LIN {X 0,Y 336.735,Z 952.723,A -85,B 0,C 180,E1 12207.175,E2 12207.175} C_VEL
LIN {X 0,Y 325.926,Z 967.689,A -85,B 0,C 180,E1 12204.691,E2 12204.691} C_VEL
LIN {X 0,Y 313.476,Z 984.143,A -85,B 0,C 180,E1 12201.395,E2 12201.395} C_VEL
LIN {X 0,Y 302.068,Z 998.366,A -85,B 0,C 180,E1 12197.857,E2 12197.857} C_VEL
LIN {X 0,Y 292.752,Z 1009.779,A -85,B 0,C 180,E1 12194.441,E2 12194.441} C_VEL
LIN {X 0,Y 282.433,Z 1022.378,A -85,B 0,C 180,E1 12189.85,E2 12189.85} C_VEL
LIN {X 0,Y 274.164,Z 1032.514,A -85,B 0,C 180,E1 12185.186,E2 12185.186} C_VEL
LIN {X 0,Y 268.041,Z 1040.43,A -85,B 0,C 180,E1 12180.734,E2 12180.734} C_VEL
LIN {X 0,Y 262.356,Z 1048.512,A -85,B 0,C 180,E1 12175.027,E2 12175.027} C_VEL
LIN {X 0,Y 258.976,Z 1054.032,A -85,B 0,C 180,E1 12169.862,E2 12169.862} C_VEL
LIN {X 0,Y 257.187,Z 1057.754,A -85,B 0,C 180,E1 12165.33,E2 12165.33} C_VEL
LIN {X 0,Y 256.255,Z 1060.464,A -85,B 0,C 180,E1 12160.795,E2 12160.795} C_VEL
LIN {X 0,Y 255.945,Z 1062.179,A -85,B 0,C 180,E1 12156.28,E2 12156.28} C_VEL
LIN {X 0,Y 255.908,Z 1062.926,A -85,B 0,C 180,E1 12151.567,E2 12151.567} C_VEL
LIN {X 0,Y 255.912,Z 1062.587,A -85,B 0,C 180,E1 12146.864,E2 12146.864} C_VEL
LIN {X 0,Y 256.04,Z 1060.822,A -85,B 0,C 180,E1 12141.692,E2 12141.692} C_VEL
LIN {X 0,Y 256.6,Z 1058.068,A -85,B 0,C 180,E1 12136.938,E2 12136.938} C_VEL
LIN {X 0,Y 257.893,Z 1054.397,A -85,B 0,C 180,E1 12132.397,E2 12132.397} C_VEL
LIN {X 0,Y 260.268,Z 1049.406,A -85,B 0,C 180,E1 12127.646,E2 12127.646} C_VEL
LIN {X 0,Y 264.917,Z 1041.534,A -85,B 0,C 180,E1 12121.85,E2 12121.85} C_VEL
LIN {X 0,Y 270.469,Z 1033.203,A -85,B 0,C 180,E1 12117.055,E2 12117.055} C_VEL
LIN {X 0,Y 277.094,Z 1023.98,A -85,B 0,C 180,E1 12112.683,E2 12112.683} C_VEL
LIN {X 0,Y 286.962,Z 1010.708,A -85,B 0,C 180,E1 12107.621,E2 12107.621} C_VEL
LIN {X 0,Y 295.813,Z 998.833,A -85,B 0,C 180,E1 12103.949,E2 12103.949} C_VEL
LIN {X 0,Y 306.537,Z 984.365,A -85,B 0,C 180,E1 12100.23,E2 12100.23} C_VEL
LIN {X 0,Y 317.721,Z 968.541,A -85,B 0,C 180,E1 12096.932,E2 12096.932} C_VEL
LIN {X 0,Y 327.989,Z 953.379,A -85,B 0,C 180,E1 12094.295,E2 12094.295} C_VEL
LIN {X 0,Y 339.558,Z 935.432,A -85,B 0,C 180,E1 12091.679,E2 12091.679} C_VEL
LIN {X 0,Y 351.058,Z 915.947,A -85,B 0,C 180,E1 12089.361,E2 12089.361} C_VEL
LIN {X 0,Y 360.57,Z 898.596,A -85,B 0,C 180,E1 12087.626,E2 12087.626} C_VEL
LIN {X 0,Y 371.142,Z 877.701,A -85,B 0,C 180,E1 12085.866,E2 12085.866} C_VEL
LIN {X 0,Y 381.228,Z 855.132,A -85,B 0,C 180,E1 12084.317,E2 12084.317} C_VEL
LIN {X 0,Y 388.946,Z 835.881,A -85,B 0,C 180,E1 12083.213,E2 12083.213} C_VEL
LIN {X 0,Y 397.181,Z 812.804,A -85,B 0,C 180,E1 12082.116,E2 12082.116} C_VEL
LIN {X 0,Y 404.562,Z 787.996,A -85,B 0,C 180,E1 12081.181,E2 12081.181} C_VEL
LIN {X 0,Y 409.672,Z 767.607,A -85,B 0,C 180,E1 12080.56,E2 12080.56} C_VEL
LIN {X 0,Y 414.754,Z 742.941,A -85,B 0,C 180,E1 12079.967,E2 12079.967} C_VEL
LIN {X 0,Y 418.524,Z 716.56,A -85,B 0,C 180,E1 12079.475,E2 12079.475} C_VEL
LIN {X 0,Y 437.682,Z 506.178,A -85,B 0,C 180,E1 12076.237,E2 12076.237} C_VEL
LIN {X 0,Y 432.715,Z 497.153,A -85,B 0,C 180,E1 12073.496,E2 12073.496} C_VEL
LIN {X 0,Y 428.974,Z 490.578,A -85,B 0,C 180,E1 12071.019,E2 12071.019} C_VEL
LIN {X 0,Y 426.712,Z 486.682,A -85,B 0,C 180,E1 12069.237,E2 12069.237} C_VEL
LIN {X 0,Y 424.543,Z 482.925,A -85,B 0,C 180,E1 12067.171,E2 12067.171} C_VEL
LIN {X 0,Y 422.269,Z 478.811,A -85,B 0,C 180,E1 12064.21,E2 12064.21} C_VEL
LIN {X 0,Y 420.494,Z 475.74,A -85,B 0,C 180,E1 12058.501,E2 12058.501} C_VEL
LIN {X 0,Y 420.904,Z 477.2,A -85,B 0,C 180,E1 12055.367,E2 12055.367} C_VEL
LIN {X 0,Y 422.548,Z 479.254,A -85,B 0,C 180,E1 12052.18,E2 12052.18} C_VEL
LIN {X 0,Y 425.298,Z 484.171,A -85,B 0,C 180,E1 12048.885,E2 12048.885} C_VEL
LIN {X 0,Y 428.058,Z 488.972,A -85,B 0,C 180,E1 12046.492,E2 12046.492} C_VEL
LIN {X 0,Y 432.057,Z 495.823,A -85,B 0,C 180,E1 12043.738,E2 12043.738} C_VEL
LIN {X 0,Y 436.565,Z 504.122,A -85,B 0,C 180,E1 12041.159,E2 12041.159} C_VEL
LIN {X 0,Y 437.639,Z 506.238,A -85,B 0,C 180,E1 12040.598,E2 12040.598} C_VEL
LIN {X 0,Y 418.656,Z 714.21,A -85,B 0,C 180,E1 12037.403,E2 12037.403} C_VEL
LIN {X 0,Y 414.746,Z 741.081,A -85,B 0,C 180,E1 12036.896,E2 12036.896} C_VEL
LIN {X 0,Y 409.832,Z 764.962,A -85,B 0,C 180,E1 12036.307,E2 12036.307} C_VEL
LIN {X 0,Y 404.496,Z 786.334,A -85,B 0,C 180,E1 12035.63,E2 12035.63} C_VEL
LIN {X 0,Y 396.755,Z 812.006,A -85,B 0,C 180,E1 12034.619,E2 12034.619} C_VEL
LIN {X 0,Y 389.497,Z 832.399,A -85,B 0,C 180,E1 12033.627,E2 12033.627} C_VEL
LIN {X 0,Y 381.614,Z 852.091,A -85,B 0,C 180,E1 12032.489,E2 12032.489} C_VEL
LIN {X 0,Y 371.507,Z 874.688,A -85,B 0,C 180,E1 12030.918,E2 12030.918} C_VEL
LIN {X 0,Y 361.031,Z 895.39,A -85,B 0,C 180,E1 12029.154,E2 12029.154} C_VEL
LIN {X 0,Y 351.198,Z 913.285,A -85,B 0,C 180,E1 12027.343,E2 12027.343} C_VEL
LIN {X 0,Y 338.52,Z 934.435,A -85,B 0,C 180,E1 12024.755,E2 12024.755} C_VEL
LIN {X 0,Y 328.196,Z 950.374,A -85,B 0,C 180,E1 12022.384,E2 12022.384} C_VEL
LIN {X 0,Y 318.152,Z 965.114,A -85,B 0,C 180,E1 12019.791,E2 12019.791} C_VEL
LIN {X 0,Y 305.579,Z 982.616,A -85,B 0,C 180,E1 12016.043,E2 12016.043} C_VEL
LIN {X 0,Y 296.17,Z 995.232,A -85,B 0,C 180,E1 12012.733,E2 12012.733} C_VEL
LIN {X 0,Y 286.879,Z 1007.573,A -85,B 0,C 180,E1 12008.856,E2 12008.856} C_VEL
LIN {X 0,Y 277.456,Z 1019.987,A -85,B 0,C 180,E1 12004.017,E2 12004.017} C_VEL
LIN {X 0,Y 271.095,Z 1028.659,A -85,B 0,C 180,E1 11999.863,E2 11999.863} C_VEL
LIN {X 0,Y 265.325,Z 1037.081,A -85,B 0,C 180,E1 11994.966,E2 11994.966} C_VEL
LIN {X 0,Y 260.629,Z 1044.701,A -85,B 0,C 180,E1 11989.265,E2 11989.265} C_VEL
LIN {X 0,Y 258.12,Z 1049.684,A -85,B 0,C 180,E1 11984.432,E2 11984.432} C_VEL
LIN {X 0,Y 256.696,Z 1053.442,A -85,B 0,C 180,E1 11979.642,E2 11979.642} C_VEL
LIN {X 0,Y 256.042,Z 1056.374,A -85,B 0,C 180,E1 11974.255,E2 11974.255} C_VEL
LIN {X 0,Y 255.923,Z 1057.688,A -85,B 0,C 180,E1 11969.328,E2 11969.328} C_VEL
LIN {X 0,Y 255.916,Z 1057.898,A -85,B 0,C 180,E1 11964.844,E2 11964.844} C_VEL
LIN {X 0,Y 256.005,Z 1057.204,A -85,B 0,C 180,E1 11960.558,E2 11960.558} C_VEL
LIN {X 0,Y 256.395,Z 1055.589,A -85,B 0,C 180,E1 11956.181,E2 11956.181} C_VEL
LIN {X 0,Y 257.427,Z 1052.964,A -85,B 0,C 180,E1 11951.662,E2 11951.662} C_VEL
LIN {X 0,Y 259.468,Z 1049.079,A -85,B 0,C 180,E1 11946.855,E2 11946.855} C_VEL
LIN {X 0,Y 263.498,Z 1042.971,A -85,B 0,C 180,E1 11941.189,E2 11941.189} C_VEL
LIN {X 0,Y 269.013,Z 1035.478,A -85,B 0,C 180,E1 11935.983,E2 11935.983} C_VEL
LIN {X 0,Y 275.246,Z 1027.677,A -85,B 0,C 180,E1 11931.597,E2 11931.597} C_VEL
LIN {X 0,Y 284.248,Z 1016.9,A -85,B 0,C 180,E1 11926.69,E2 11926.69} C_VEL
LIN {X 0,Y 294.039,Z 1005.111,A -85,B 0,C 180,E1 11922.446,E2 11922.446} C_VEL
LIN {X 0,Y 303.724,Z 993.402,A -85,B 0,C 180,E1 11918.961,E2 11918.961} C_VEL
LIN {X 0,Y 316.508,Z 977.44,A -85,B 0,C 180,E1 11915.094,E2 11915.094} C_VEL
LIN {X 0,Y 327.49,Z 962.979,A -85,B 0,C 180,E1 11912.25,E2 11912.25} C_VEL
LIN {X 0,Y 338.542,Z 947.715,A -85,B 0,C 180,E1 11909.735,E2 11909.735} C_VEL
LIN {X 0,Y 352.289,Z 927.25,A -85,B 0,C 180,E1 11906.974,E2 11906.974} C_VEL
LIN {X 0,Y 362.606,Z 910.598,A -85,B 0,C 180,E1 11905.129,E2 11905.129} C_VEL
LIN {X 0,Y 372.78,Z 892.869,A -85,B 0,C 180,E1 11903.462,E2 11903.462} C_VEL
LIN {X 0,Y 384.665,Z 869.928,A -85,B 0,C 180,E1 11901.678,E2 11901.678} C_VEL
LIN {X 0,Y 393.697,Z 850.323,A -85,B 0,C 180,E1 11900.42,E2 11900.42} C_VEL
LIN {X 0,Y 402.231,Z 829.664,A -85,B 0,C 180,E1 11899.306,E2 11899.306} C_VEL
LIN {X 0,Y 411.481,Z 803.641,A -85,B 0,C 180,E1 11898.174,E2 11898.174} C_VEL
LIN {X 0,Y 417.687,Z 783.031,A -85,B 0,C 180,E1 11897.455,E2 11897.455} C_VEL
LIN {X 0,Y 423.053,Z 761.928,A -85,B 0,C 180,E1 11896.847,E2 11896.847} C_VEL
LIN {X 0,Y 428.658,Z 733.815,A -85,B 0,C 180,E1 11896.229,E2 11896.229} C_VEL
LIN {X 0,Y 431.2,Z 716.612,A -85,B 0,C 180,E1 11895.925,E2 11895.925} C_VEL
LIN {X 0,Y 431.767,Z 709.092,A -85,B 0,C 180,E1 11895.676,E2 11895.676} C_VEL
LIN {X 0,Y 431.958,Z 689.518,A -85,B 0,C 180,E1 11894.578,E2 11894.578} C_VEL
LIN {X 0,Y 432.363,Z 683.031,A -85,B 0,C 180,E1 11894.388,E2 11894.388} C_VEL
LIN {X 0,Y 448.077,Z 521.035,A -85,B 0,C 180,E1 11891.978,E2 11891.978} C_VEL
LIN {X 0,Y 444.633,Z 514.491,A -85,B 0,C 180,E1 11889.449,E2 11889.449} C_VEL
LIN {X 0,Y 442.12,Z 509.966,A -85,B 0,C 180,E1 11887.145,E2 11887.145} C_VEL
LIN {X 0,Y 440.219,Z 506.351,A -85,B 0,C 180,E1 11884.821,E2 11884.821} C_VEL
LIN {X 0,Y 438.336,Z 501.994,A -85,B 0,C 180,E1 11880.392,E2 11880.392} C_VEL
LIN {X 0,Y 438.418,Z 502.124,A -85,B 0,C 180,E1 11876.339,E2 11876.339} C_VEL
LIN {X 0,Y 440.195,Z 506.386,A -85,B 0,C 180,E1 11872.298,E2 11872.298} C_VEL
LIN {X 0,Y 441.119,Z 508.161,A -85,B 0,C 180,E1 11871.068,E2 11871.068} C_VEL
LIN {X 0,Y 443.036,Z 511.664,A -85,B 0,C 180,E1 11869.037,E2 11869.037} C_VEL
LIN {X 0,Y 445.731,Z 516.615,A -85,B 0,C 180,E1 11866.773,E2 11866.773} C_VEL
LIN {X 0,Y 448.131,Z 521.442,A -85,B 0,C 180,E1 11865.061,E2 11865.061} C_VEL
LIN {X 0,Y 428.944,Z 716.865,A -85,B 0,C 180,E1 11862.164,E2 11862.164} C_VEL
LIN {X 0,Y 424.778,Z 743.872,A -85,B 0,C 180,E1 11861.688,E2 11861.688} C_VEL
LIN {X 0,Y 419.625,Z 767.55,A -85,B 0,C 180,E1 11861.159,E2 11861.159} C_VEL
LIN {X 0,Y 414.229,Z 787.872,A -85,B 0,C 180,E1 11860.595,E2 11860.595} C_VEL
LIN {X 0,Y 406.633,Z 812.077,A -85,B 0,C 180,E1 11859.757,E2 11859.757} C_VEL
LIN {X 0,Y 398.007,Z 834.964,A -85,B 0,C 180,E1 11858.755,E2 11858.755} C_VEL
LIN {X 0,Y 389.986,Z 853.879,A -85,B 0,C 180,E1 11857.754,E2 11857.754} C_VEL
LIN {X 0,Y 380.517,Z 873.928,A -85,B 0,C 180,E1 11856.501,E2 11856.501} C_VEL
LIN {X 0,Y 368.599,Z 896.322,A -85,B 0,C 180,E1 11854.793,E2 11854.793} C_VEL
LIN {X 0,Y 358.091,Z 914.215,A -85,B 0,C 180,E1 11853.142,E2 11853.142} C_VEL
LIN {X 0,Y 346.16,Z 933.011,A -85,B 0,C 180,E1 11851.071,E2 11851.071} C_VEL
LIN {X 0,Y 332.963,Z 951.98,A -85,B 0,C 180,E1 11848.498,E2 11848.498} C_VEL
LIN {X 0,Y 321.859,Z 966.938,A -85,B 0,C 180,E1 11846.043,E2 11846.043} C_VEL
LIN {X 0,Y 309.548,Z 982.746,A -85,B 0,C 180,E1 11842.925,E2 11842.925} C_VEL
LIN {X 0,Y 297.095,Z 997.78,A -85,B 0,C 180,E1 11839.222,E2 11839.222} C_VEL
LIN {X 0,Y 287.355,Z 1009.241,A -85,B 0,C 180,E1 11835.791,E2 11835.791} C_VEL
LIN {X 0,Y 276.791,Z 1021.62,A -85,B 0,C 180,E1 11831.289,E2 11831.289} C_VEL
LIN {X 0,Y 267.758,Z 1032.109,A -85,B 0,C 180,E1 11826.424,E2 11826.424} C_VEL
LIN {X 0,Y 261.207,Z 1040.066,A -85,B 0,C 180,E1 11821.888,E2 11821.888} C_VEL
LIN {X 0,Y 255.228,Z 1048.032,A -85,B 0,C 180,E1 11816.215,E2 11816.215} C_VEL
LIN {X 0,Y 251.264,Z 1053.993,A -85,B 0,C 180,E1 11810.499,E2 11810.499} C_VEL
LIN {X 0,Y 249.25,Z 1057.866,A -85,B 0,C 180,E1 11805.591,E2 11805.591} C_VEL
LIN {X 0,Y 248.234,Z 1060.661,A -85,B 0,C 180,E1 11800.629,E2 11800.629} C_VEL
LIN {X 0,Y 247.917,Z 1062.458,A -85,B 0,C 180,E1 11795.323,E2 11795.323} C_VEL
LIN {X 0,Y 247.927,Z 1062.847,A -85,B 0,C 180,E1 11790.231,E2 11790.231} C_VEL
LIN {X 0,Y 247.909,Z 1062.171,A -85,B 0,C 180,E1 11785.605,E2 11785.605} C_VEL
LIN {X 0,Y 248.062,Z 1060.606,A -85,B 0,C 180,E1 11781.189,E2 11781.189} C_VEL
LIN {X 0,Y 248.68,Z 1057.958,A -85,B 0,C 180,E1 11776.514,E2 11776.514} C_VEL
LIN {X 0,Y 250.09,Z 1054.277,A -85,B 0,C 180,E1 11771.829,E2 11771.829} C_VEL
LIN {X 0,Y 252.654,Z 1049.276,A -85,B 0,C 180,E1 11766.934,E2 11766.934} C_VEL
LIN {X 0,Y 257.86,Z 1041.018,A -85,B 0,C 180,E1 11760.748,E2 11760.748} C_VEL
LIN {X 0,Y 263.472,Z 1033.085,A -85,B 0,C 180,E1 11756.092,E2 11756.092} C_VEL
LIN {X 0,Y 270.136,Z 1024.272,A -85,B 0,C 180,E1 11751.82,E2 11751.82} C_VEL
LIN {X 0,Y 279.766,Z 1011.932,A -85,B 0,C 180,E1 11746.95,E2 11746.95} C_VEL
LIN {X 0,Y 289.577,Z 999.267,A -85,B 0,C 180,E1 11742.944,E2 11742.944} C_VEL
LIN {X 0,Y 299.517,Z 986.31,A -85,B 0,C 180,E1 11739.543,E2 11739.543} C_VEL
LIN {X 0,Y 312.183,Z 969.143,A -85,B 0,C 180,E1 11735.872,E2 11735.872} C_VEL
LIN {X 0,Y 322.736,Z 954.047,A -85,B 0,C 180,E1 11733.228,E2 11733.228} C_VEL
LIN {X 0,Y 333.46,Z 937.893,A -85,B 0,C 180,E1 11730.847,E2 11730.847} C_VEL
LIN {X 0,Y 346.371,Z 916.849,A -85,B 0,C 180,E1 11728.303,E2 11728.303} C_VEL
LIN {X 0,Y 356.09,Z 899.594,A -85,B 0,C 180,E1 11726.577,E2 11726.577} C_VEL
LIN {X 0,Y 365.881,Z 880.749,A -85,B 0,C 180,E1 11724.98,E2 11724.98} C_VEL
LIN {X 0,Y 377.235,Z 856.32,A -85,B 0,C 180,E1 11723.285,E2 11723.285} C_VEL
LIN {X 0,Y 385.404,Z 836.41,A -85,B 0,C 180,E1 11722.151,E2 11722.151} C_VEL
LIN {X 0,Y 393.112,Z 815.314,A -85,B 0,C 180,E1 11721.154,E2 11721.154} C_VEL
LIN {X 0,Y 401.068,Z 789.631,A -85,B 0,C 180,E1 11720.177,E2 11720.177} C_VEL
LIN {X 0,Y 406.458,Z 768.682,A -85,B 0,C 180,E1 11719.54,E2 11719.54} C_VEL
LIN {X 0,Y 411.248,Z 746.109,A -85,B 0,C 180,E1 11718.997,E2 11718.997} C_VEL
LIN {X 0,Y 415.567,Z 717.905,A -85,B 0,C 180,E1 11718.465,E2 11718.465} C_VEL
LIN {X 0,Y 425.663,Z 609.9,A -85,B 0,C 180,E1 11716.798,E2 11716.798} C_VEL
LIN {X 0,Y 434.788,Z 511.445,A -85,B 0,C 180,E1 11715.301,E2 11715.301} C_VEL
LIN {X 0,Y 430.262,Z 502.918,A -85,B 0,C 180,E1 11712.618,E2 11712.618} C_VEL
LIN {X 0,Y 426.048,Z 495.294,A -85,B 0,C 180,E1 11709.524,E2 11709.524} C_VEL
LIN {X 0,Y 423.304,Z 490.638,A -85,B 0,C 180,E1 11706.919,E2 11706.919} C_VEL
LIN {X 0,Y 421.203,Z 486.697,A -85,B 0,C 180,E1 11704.084,E2 11704.084} C_VEL
LIN {X 0,Y 419.519,Z 483.683,A -85,B 0,C 180,E1 11698.498,E2 11698.498} C_VEL
LIN {X 0,Y 420.018,Z 485.34,A -85,B 0,C 180,E1 11695.084,E2 11695.084} C_VEL
LIN {X 0,Y 421.476,Z 487.179,A -85,B 0,C 180,E1 11692.297,E2 11692.297} C_VEL
LIN {X 0,Y 424.108,Z 492.007,A -85,B 0,C 180,E1 11689.059,E2 11689.059} C_VEL
LIN {X 0,Y 426.729,Z 496.681,A -85,B 0,C 180,E1 11686.725,E2 11686.725} C_VEL
LIN {X 0,Y 430.589,Z 503.495,A -85,B 0,C 180,E1 11683.993,E2 11683.993} C_VEL
LIN {X 0,Y 434.769,Z 511.39,A -85,B 0,C 180,E1 11681.53,E2 11681.53} C_VEL
LIN {X 0,Y 415.857,Z 714.241,A -85,B 0,C 180,E1 11678.435,E2 11678.435} C_VEL
LIN {X 0,Y 411.897,Z 741.045,A -85,B 0,C 180,E1 11677.936,E2 11677.936} C_VEL
LIN {X 0,Y 406.891,Z 765,A -85,B 0,C 180,E1 11677.356,E2 11677.356} C_VEL
LIN {X 0,Y 401.415,Z 786.552,A -85,B 0,C 180,E1 11676.684,E2 11676.684} C_VEL
LIN {X 0,Y 393.637,Z 811.908,A -85,B 0,C 180,E1 11675.701,E2 11675.701} C_VEL
LIN {X 0,Y 386.006,Z 832.931,A -85,B 0,C 180,E1 11674.692,E2 11674.692} C_VEL
LIN {X 0,Y 377.974,Z 852.577,A -85,B 0,C 180,E1 11673.567,E2 11673.567} C_VEL
LIN {X 0,Y 367.135,Z 876.128,A -85,B 0,C 180,E1 11671.934,E2 11671.934} C_VEL
LIN {X 0,Y 356.959,Z 895.772,A -85,B 0,C 180,E1 11670.267,E2 11670.267} C_VEL
LIN {X 0,Y 347.096,Z 913.3,A -85,B 0,C 180,E1 11668.505,E2 11668.505} C_VEL
LIN {X 0,Y 334.232,Z 934.247,A -85,B 0,C 180,E1 11665.962,E2 11665.962} C_VEL
LIN {X 0,Y 323.726,Z 950.04,A -85,B 0,C 180,E1 11663.627,E2 11663.627} C_VEL
LIN {X 0,Y 313.458,Z 964.67,A -85,B 0,C 180,E1 11661.067,E2 11661.067} C_VEL
LIN {X 0,Y 301.039,Z 981.477,A -85,B 0,C 180,E1 11657.507,E2 11657.507} C_VEL
LIN {X 0,Y 290.692,Z 994.835,A -85,B 0,C 180,E1 11654.012,E2 11654.012} C_VEL
LIN {X 0,Y 281.403,Z 1006.657,A -85,B 0,C 180,E1 11650.292,E2 11650.292} C_VEL
LIN {X 0,Y 270.976,Z 1019.83,A -85,B 0,C 180,E1 11645.144,E2 11645.144} C_VEL
LIN {X 0,Y 263.942,Z 1028.944,A -85,B 0,C 180,E1 11640.689,E2 11640.689} C_VEL
LIN {X 0,Y 257.713,Z 1037.593,A -85,B 0,C 180,E1 11635.509,E2 11635.509} C_VEL
LIN {X 0,Y 252.903,Z 1044.938,A -85,B 0,C 180,E1 11629.784,E2 11629.784} C_VEL
LIN {X 0,Y 250.347,Z 1049.677,A -85,B 0,C 180,E1 11625.047,E2 11625.047} C_VEL
LIN {X 0,Y 248.806,Z 1053.4,A -85,B 0,C 180,E1 11620.185,E2 11620.185} C_VEL
LIN {X 0,Y 248.065,Z 1056.377,A -85,B 0,C 180,E1 11614.624,E2 11614.624} C_VEL
LIN {X 0,Y 247.922,Z 1057.771,A -85,B 0,C 180,E1 11609.307,E2 11609.307} C_VEL
LIN {X 0,Y 247.92,Z 1057.971,A -85,B 0,C 180,E1 11604.677,E2 11604.677} C_VEL
LIN {X 0,Y 248.023,Z 1057.266,A -85,B 0,C 180,E1 11600.252,E2 11600.252} C_VEL
LIN {X 0,Y 248.492,Z 1055.557,A -85,B 0,C 180,E1 11595.553,E2 11595.553} C_VEL
LIN {X 0,Y 249.69,Z 1052.846,A -85,B 0,C 180,E1 11590.83,E2 11590.83} C_VEL
LIN {X 0,Y 252.129,Z 1048.698,A -85,B 0,C 180,E1 11585.642,E2 11585.642} C_VEL
LIN {X 0,Y 257.058,Z 1041.766,A -85,B 0,C 180,E1 11579.366,E2 11579.366} C_VEL
LIN {X 0,Y 262.541,Z 1034.899,A -85,B 0,C 180,E1 11574.59,E2 11574.59} C_VEL
LIN {X 0,Y 270.146,Z 1026.037,A -85,B 0,C 180,E1 11569.63,E2 11569.63} C_VEL
LIN {X 0,Y 279.915,Z 1014.789,A -85,B 0,C 180,E1 11564.696,E2 11564.696} C_VEL
LIN {X 0,Y 289.414,Z 1003.903,A -85,B 0,C 180,E1 11560.833,E2 11560.833} C_VEL
LIN {X 0,Y 301.181,Z 990.25,A -85,B 0,C 180,E1 11556.861,E2 11556.861} C_VEL
LIN {X 0,Y 313.573,Z 975.01,A -85,B 0,C 180,E1 11553.339,E2 11553.339} C_VEL
LIN {X 0,Y 324.392,Z 961.157,A -85,B 0,C 180,E1 11550.687,E2 11550.687} C_VEL
LIN {X 0,Y 337.579,Z 943.278,A -85,B 0,C 180,E1 11547.855,E2 11547.855} C_VEL
LIN {X 0,Y 349.444,Z 925.75,A -85,B 0,C 180,E1 11545.599,E2 11545.599} C_VEL
LIN {X 0,Y 360.039,Z 908.951,A -85,B 0,C 180,E1 11543.784,E2 11543.784} C_VEL
LIN {X 0,Y 371.888,Z 888.56,A -85,B 0,C 180,E1 11541.938,E2 11541.938} C_VEL
LIN {X 0,Y 382.89,Z 867.179,A -85,B 0,C 180,E1 11540.364,E2 11540.364} C_VEL
LIN {X 0,Y 391.262,Z 849.205,A -85,B 0,C 180,E1 11539.249,E2 11539.249} C_VEL
LIN {X 0,Y 400.715,Z 826.557,A -85,B 0,C 180,E1 11538.068,E2 11538.068} C_VEL
LIN {X 0,Y 409.008,Z 803.134,A -85,B 0,C 180,E1 11537.087,E2 11537.087} C_VEL
LIN {X 0,Y 415.36,Z 782.286,A -85,B 0,C 180,E1 11536.379,E2 11536.379} C_VEL
LIN {X 0,Y 420.957,Z 760.479,A -85,B 0,C 180,E1 11535.772,E2 11535.772} C_VEL
LIN {X 0,Y 426.355,Z 733.373,A -85,B 0,C 180,E1 11535.194,E2 11535.194} C_VEL
LIN {X 0,Y 429.535,Z 710.871,A -85,B 0,C 180,E1 11534.81,E2 11534.81} C_VEL
LIN {X 0,Y 432.363,Z 683.031,A -85,B 0,C 180,E1 11534.388,E2 11534.388} C_VEL
LIN {X 0,Y 432.821,Z 675.49,A -85,B 0,C 180,E1 11534.151,E2 11534.151} C_VEL
LIN {X 0,Y 433.079,Z 655.91,A -85,B 0,C 180,E1 11533.058,E2 11533.058} C_VEL
LIN {X 0,Y 433.524,Z 649.426,A -85,B 0,C 180,E1 11532.865,E2 11532.865} C_VEL
LIN {X 0,Y 445.692,Z 526.793,A -85,B 0,C 180,E1 11531.059,E2 11531.059} C_VEL
LIN {X 0,Y 442.72,Z 521.185,A -85,B 0,C 180,E1 11528.704,E2 11528.704} C_VEL
LIN {X 0,Y 440.885,Z 517.666,A -85,B 0,C 180,E1 11526.904,E2 11526.904} C_VEL
LIN {X 0,Y 439.146,Z 514.228,A -85,B 0,C 180,E1 11524.702,E2 11524.702} C_VEL
LIN {X 0,Y 437.332,Z 509.914,A -85,B 0,C 180,E1 11520.262,E2 11520.262} C_VEL
LIN {X 0,Y 437.431,Z 510.173,A -85,B 0,C 180,E1 11516.33,E2 11516.33} C_VEL
LIN {X 0,Y 439.222,Z 514.373,A -85,B 0,C 180,E1 11512.281,E2 11512.281} C_VEL
LIN {X 0,Y 441.682,Z 519.144,A -85,B 0,C 180,E1 11509.368,E2 11509.368} C_VEL
LIN {X 0,Y 444.485,Z 524.476,A -85,B 0,C 180,E1 11506.934,E2 11506.934} C_VEL
LIN {X 0,Y 445.73,Z 527.273,A -85,B 0,C 180,E1 11505.979,E2 11505.979} C_VEL
LIN {X 0,Y 426.748,Z 716.79,A -85,B 0,C 180,E1 11503.199,E2 11503.199} C_VEL
LIN {X 0,Y 422.531,Z 743.731,A -85,B 0,C 180,E1 11502.731,E2 11502.731} C_VEL
LIN {X 0,Y 417.305,Z 767.42,A -85,B 0,C 180,E1 11502.215,E2 11502.215} C_VEL
LIN {X 0,Y 411.858,Z 787.635,A -85,B 0,C 180,E1 11501.668,E2 11501.668} C_VEL
LIN {X 0,Y 403.908,Z 812.509,A -85,B 0,C 180,E1 11500.822,E2 11500.822} C_VEL
LIN {X 0,Y 395.164,Z 835.291,A -85,B 0,C 180,E1 11499.841,E2 11499.841} C_VEL
LIN {X 0,Y 386.599,Z 855.059,A -85,B 0,C 180,E1 11498.809,E2 11498.809} C_VEL
LIN {X 0,Y 375.78,Z 877.325,A -85,B 0,C 180,E1 11497.414,E2 11497.414} C_VEL
LIN {X 0,Y 364.407,Z 897.891,A -85,B 0,C 180,E1 11495.83,E2 11495.83} C_VEL
LIN {X 0,Y 354.102,Z 914.988,A -85,B 0,C 180,E1 11494.259,E2 11494.259} C_VEL
LIN {X 0,Y 341.189,Z 934.784,A -85,B 0,C 180,E1 11492.076,E2 11492.076} C_VEL
LIN {X 0,Y 328.099,Z 952.94,A -85,B 0,C 180,E1 11489.592,E2 11489.592} C_VEL
LIN {X 0,Y 316.668,Z 967.872,A -85,B 0,C 180,E1 11487.13,E2 11487.13} C_VEL
LIN {X 0,Y 302.799,Z 984.964,A -85,B 0,C 180,E1 11483.68,E2 11483.68} C_VEL
LIN {X 0,Y 291.18,Z 998.461,A -85,B 0,C 180,E1 11480.282,E2 11480.282} C_VEL
LIN {X 0,Y 281.114,Z 1009.848,A -85,B 0,C 180,E1 11476.816,E2 11476.816} C_VEL
LIN {X 0,Y 269.864,Z 1022.4,A -85,B 0,C 180,E1 11472.116,E2 11472.116} C_VEL
LIN {X 0,Y 260.743,Z 1032.515,A -85,B 0,C 180,E1 11467.293,E2 11467.293} C_VEL
LIN {X 0,Y 253.705,Z 1040.649,A -85,B 0,C 180,E1 11462.498,E2 11462.498} C_VEL
LIN {X 0,Y 247.058,Z 1048.962,A -85,B 0,C 180,E1 11456.177,E2 11456.177} C_VEL
LIN {X 0,Y 243.447,Z 1054.161,A -85,B 0,C 180,E1 11450.936,E2 11450.936} C_VEL
LIN {X 0,Y 241.318,Z 1057.979,A -85,B 0,C 180,E1 11445.871,E2 11445.871} C_VEL
LIN {X 0,Y 240.172,Z 1061.039,A -85,B 0,C 180,E1 11440.07,E2 11440.07} C_VEL
LIN {X 0,Y 239.91,Z 1062.475,A -85,B 0,C 180,E1 11434.782,E2 11434.782} C_VEL
LIN {X 0,Y 239.937,Z 1062.742,A -85,B 0,C 180,E1 11430,E2 11430} C_VEL
LIN {X 0,Y 239.911,Z 1062.08,A -85,B 0,C 180,E1 11425.458,E2 11425.458} C_VEL
LIN {X 0,Y 240.086,Z 1060.445,A -85,B 0,C 180,E1 11420.766,E2 11420.766} C_VEL
LIN {X 0,Y 240.768,Z 1057.848,A -85,B 0,C 180,E1 11416.062,E2 11416.062} C_VEL
LIN {X 0,Y 242.305,Z 1054.157,A -85,B 0,C 180,E1 11411.224,E2 11411.224} C_VEL
LIN {X 0,Y 245.242,Z 1048.887,A -85,B 0,C 180,E1 11405.939,E2 11405.939} C_VEL
LIN {X 0,Y 250.896,Z 1040.516,A -85,B 0,C 180,E1 11399.594,E2 11399.594} C_VEL
LIN {X 0,Y 256.951,Z 1032.465,A -85,B 0,C 180,E1 11394.805,E2 11394.805} C_VEL
LIN {X 0,Y 265.185,Z 1022.239,A -85,B 0,C 180,E1 11389.853,E2 11389.853} C_VEL
LIN {X 0,Y 275.215,Z 1009.843,A -85,B 0,C 180,E1 11385.11,E2 11385.11} C_VEL
LIN {X 0,Y 284.471,Z 998.413,A -85,B 0,C 180,E1 11381.525,E2 11381.525} C_VEL
LIN {X 0,Y 296.001,Z 983.957,A -85,B 0,C 180,E1 11377.773,E2 11377.773} C_VEL
LIN {X 0,Y 308.421,Z 967.441,A -85,B 0,C 180,E1 11374.34,E2 11374.34} C_VEL
LIN {X 0,Y 318.913,Z 952.84,A -85,B 0,C 180,E1 11371.825,E2 11371.825} C_VEL
LIN {X 0,Y 331.148,Z 934.856,A -85,B 0,C 180,E1 11369.236,E2 11369.236} C_VEL
LIN {X 0,Y 343.252,Z 915.289,A -85,B 0,C 180,E1 11366.954,E2 11366.954} C_VEL
LIN {X 0,Y 353.232,Z 897.892,A -85,B 0,C 180,E1 11365.258,E2 11365.258} C_VEL
LIN {X 0,Y 364.282,Z 876.941,A -85,B 0,C 180,E1 11363.543,E2 11363.543} C_VEL
LIN {X 0,Y 374.431,Z 855.054,A -85,B 0,C 180,E1 11362.085,E2 11362.085} C_VEL
LIN {X 0,Y 382.398,Z 835.919,A -85,B 0,C 180,E1 11361.017,E2 11361.017} C_VEL
LIN {X 0,Y 390.926,Z 812.866,A -85,B 0,C 180,E1 11359.954,E2 11359.954} C_VEL
LIN {X 0,Y 398.542,Z 788.202,A -85,B 0,C 180,E1 11359.054,E2 11359.054} C_VEL
LIN {X 0,Y 403.82,Z 767.905,A -85,B 0,C 180,E1 11358.457,E2 11358.457} C_VEL
LIN {X 0,Y 408.852,Z 744.355,A -85,B 0,C 180,E1 11357.906,E2 11357.906} C_VEL
LIN {X 0,Y 412.976,Z 717.187,A -85,B 0,C 180,E1 11357.407,E2 11357.407} C_VEL
LIN {X 0,Y 428.466,Z 554.319,A -85,B 0,C 180,E1 11354.934,E2 11354.934} C_VEL
LIN {X 0,Y 432.023,Z 516.757,A -85,B 0,C 180,E1 11354.362,E2 11354.362} C_VEL
LIN {X 0,Y 427.6,Z 508.423,A -85,B 0,C 180,E1 11351.533,E2 11351.533} C_VEL
LIN {X 0,Y 424.191,Z 502.167,A -85,B 0,C 180,E1 11348.813,E2 11348.813} C_VEL
LIN {X 0,Y 422.073,Z 498.349,A -85,B 0,C 180,E1 11346.666,E2 11346.666} C_VEL
LIN {X 0,Y 420.139,Z 494.584,A -85,B 0,C 180,E1 11343.958,E2 11343.958} C_VEL
LIN {X 0,Y 418.543,Z 491.629,A -85,B 0,C 180,E1 11338.357,E2 11338.357} C_VEL
LIN {X 0,Y 420.294,Z 494.762,A -85,B 0,C 180,E1 11332.619,E2 11332.619} C_VEL
LIN {X 0,Y 422.922,Z 499.84,A -85,B 0,C 180,E1 11329.235,E2 11329.235} C_VEL
LIN {X 0,Y 425.407,Z 504.389,A -85,B 0,C 180,E1 11326.959,E2 11326.959} C_VEL
LIN {X 0,Y 429.13,Z 511.167,A -85,B 0,C 180,E1 11324.249,E2 11324.249} C_VEL
LIN {X 0,Y 431.996,Z 516.87,A -85,B 0,C 180,E1 11322.464,E2 11322.464} C_VEL
LIN {X 0,Y 413.186,Z 714.338,A -85,B 0,C 180,E1 11319.48,E2 11319.48} C_VEL
LIN {X 0,Y 409.139,Z 741.239,A -85,B 0,C 180,E1 11318.986,E2 11318.986} C_VEL
LIN {X 0,Y 404.062,Z 765.146,A -85,B 0,C 180,E1 11318.416,E2 11318.416} C_VEL
LIN {X 0,Y 398.59,Z 786.343,A -85,B 0,C 180,E1 11317.767,E2 11317.767} C_VEL
LIN {X 0,Y 390.972,Z 810.938,A -85,B 0,C 180,E1 11316.838,E2 11316.838} C_VEL
LIN {X 0,Y 383.041,Z 832.466,A -85,B 0,C 180,E1 11315.829,E2 11315.829} C_VEL
LIN {X 0,Y 374.856,Z 852.171,A -85,B 0,C 180,E1 11314.721,E2 11314.721} C_VEL
LIN {X 0,Y 364.176,Z 875.087,A -85,B 0,C 180,E1 11313.166,E2 11313.166} C_VEL
LIN {X 0,Y 353.393,Z 895.495,A -85,B 0,C 180,E1 11311.465,E2 11311.465} C_VEL
LIN {X 0,Y 343.542,Z 912.636,A -85,B 0,C 180,E1 11309.766,E2 11309.766} C_VEL
LIN {X 0,Y 331.123,Z 932.555,A -85,B 0,C 180,E1 11307.404,E2 11307.404} C_VEL
LIN {X 0,Y 319.168,Z 950.047,A -85,B 0,C 180,E1 11304.851,E2 11304.851} C_VEL
LIN {X 0,Y 308.479,Z 964.831,A -85,B 0,C 180,E1 11302.268,E2 11302.268} C_VEL
LIN {X 0,Y 295.576,Z 981.719,A -85,B 0,C 180,E1 11298.676,E2 11298.676} C_VEL
LIN {X 0,Y 284.856,Z 995.063,A -85,B 0,C 180,E1 11295.157,E2 11295.157} C_VEL
LIN {X 0,Y 275.197,Z 1006.872,A -85,B 0,C 180,E1 11291.396,E2 11291.396} C_VEL
LIN {X 0,Y 264.701,Z 1019.566,A -85,B 0,C 180,E1 11286.374,E2 11286.374} C_VEL
LIN {X 0,Y 257.33,Z 1028.611,A -85,B 0,C 180,E1 11281.9,E2 11281.9} C_VEL
LIN {X 0,Y 251.092,Z 1036.712,A -85,B 0,C 180,E1 11276.998,E2 11276.998} C_VEL
LIN {X 0,Y 245.49,Z 1044.73,A -85,B 0,C 180,E1 11270.754,E2 11270.754} C_VEL
LIN {X 0,Y 242.638,Z 1049.601,A -85,B 0,C 180,E1 11265.782,E2 11265.782} C_VEL
LIN {X 0,Y 241.002,Z 1053.201,A -85,B 0,C 180,E1 11261.002,E2 11261.002} C_VEL
LIN {X 0,Y 240.163,Z 1055.92,A -85,B 0,C 180,E1 11255.974,E2 11255.974} C_VEL
LIN {X 0,Y 239.948,Z 1057.709,A -85,B 0,C 180,E1 11250.477,E2 11250.477} C_VEL
LIN {X 0,Y 239.914,Z 1058.11,A -85,B 0,C 180,E1 11245.219,E2 11245.219} C_VEL
LIN {X 0,Y 240.029,Z 1057.396,A -85,B 0,C 180,E1 11240.166,E2 11240.166} C_VEL
LIN {X 0,Y 240.531,Z 1055.722,A -85,B 0,C 180,E1 11235.311,E2 11235.311} C_VEL
LIN {X 0,Y 241.815,Z 1053.047,A -85,B 0,C 180,E1 11230.432,E2 11230.432} C_VEL
LIN {X 0,Y 244.262,Z 1049.141,A -85,B 0,C 180,E1 11225.321,E2 11225.321} C_VEL
LIN {X 0,Y 249.165,Z 1042.684,A -85,B 0,C 180,E1 11219.092,E2 11219.092} C_VEL
LIN {X 0,Y 255.06,Z 1035.652,A -85,B 0,C 180,E1 11213.983,E2 11213.983} C_VEL
LIN {X 0,Y 262.082,Z 1027.811,A -85,B 0,C 180,E1 11209.396,E2 11209.396} C_VEL
LIN {X 0,Y 272.2,Z 1016.814,A -85,B 0,C 180,E1 11204.25,E2 11204.25} C_VEL
LIN {X 0,Y 282.92,Z 1004.999,A -85,B 0,C 180,E1 11199.923,E2 11199.923} C_VEL
LIN {X 0,Y 293.617,Z 993.036,A -85,B 0,C 180,E1 11196.338,E2 11196.338} C_VEL
LIN {X 0,Y 307.362,Z 976.956,A -85,B 0,C 180,E1 11192.464,E2 11192.464} C_VEL
LIN {X 0,Y 318.849,Z 962.741,A -85,B 0,C 180,E1 11189.698,E2 11189.698} C_VEL
LIN {X 0,Y 330.901,Z 946.991,A -85,B 0,C 180,E1 11187.147,E2 11187.147} C_VEL
LIN {X 0,Y 344.684,Z 927.449,A -85,B 0,C 180,E1 11184.574,E2 11184.574} C_VEL
LIN {X 0,Y 355.624,Z 910.588,A -85,B 0,C 180,E1 11182.748,E2 11182.748} C_VEL
LIN {X 0,Y 366.51,Z 892.41,A -85,B 0,C 180,E1 11181.09,E2 11181.09} C_VEL
LIN {X 0,Y 378.791,Z 869.545,A -85,B 0,C 180,E1 11179.377,E2 11179.377} C_VEL
LIN {X 0,Y 387.907,Z 850.475,A -85,B 0,C 180,E1 11178.197,E2 11178.197} C_VEL
LIN {X 0,Y 396.573,Z 830.232,A -85,B 0,C 180,E1 11177.142,E2 11177.142} C_VEL
LIN {X 0,Y 406.263,Z 803.927,A -85,B 0,C 180,E1 11176.036,E2 11176.036} C_VEL
LIN {X 0,Y 412.668,Z 783.34,A -85,B 0,C 180,E1 11175.346,E2 11175.346} C_VEL
LIN {X 0,Y 418.063,Z 762.841,A -85,B 0,C 180,E1 11174.778,E2 11174.778} C_VEL
LIN {X 0,Y 423.722,Z 735.82,A -85,B 0,C 180,E1 11174.198,E2 11174.198} C_VEL
LIN {X 0,Y 427.197,Z 712.145,A -85,B 0,C 180,E1 11173.798,E2 11173.798} C_VEL
LIN {X 0,Y 433.524,Z 649.426,A -85,B 0,C 180,E1 11172.865,E2 11172.865} C_VEL
LIN {X 0,Y 434.02,Z 641.889,A -85,B 0,C 180,E1 11172.627,E2 11172.627} C_VEL
LIN {X 0,Y 434.5,Z 622.311,A -85,B 0,C 180,E1 11171.539,E2 11171.539} C_VEL
LIN {X 0,Y 434.982,Z 615.83,A -85,B 0,C 180,E1 11171.347,E2 11171.347} C_VEL
LIN {X 0,Y 443.411,Z 532.673,A -85,B 0,C 180,E1 11170.131,E2 11170.131} C_VEL
LIN {X 0,Y 440.152,Z 526.116,A -85,B 0,C 180,E1 11167.178,E2 11167.178} C_VEL
LIN {X 0,Y 437.983,Z 522.001,A -85,B 0,C 180,E1 11164.452,E2 11164.452} C_VEL
LIN {X 0,Y 436.356,Z 517.856,A -85,B 0,C 180,E1 11160.263,E2 11160.263} C_VEL
LIN {X 0,Y 436.426,Z 518.059,A -85,B 0,C 180,E1 11156.453,E2 11156.453} C_VEL
LIN {X 0,Y 438.154,Z 522.255,A -85,B 0,C 180,E1 11152.394,E2 11152.394} C_VEL
LIN {X 0,Y 440.497,Z 526.983,A -85,B 0,C 180,E1 11149.537,E2 11149.537} C_VEL
LIN {X 0,Y 443.162,Z 532.181,A -85,B 0,C 180,E1 11147.159,E2 11147.159} C_VEL
LIN {X 0,Y 443.458,Z 532.985,A -85,B 0,C 180,E1 11146.909,E2 11146.909} C_VEL
LIN {X 0,Y 424.692,Z 716.716,A -85,B 0,C 180,E1 11144.244,E2 11144.244} C_VEL
LIN {X 0,Y 420.399,Z 743.719,A -85,B 0,C 180,E1 11143.783,E2 11143.783} C_VEL
LIN {X 0,Y 415.127,Z 767.29,A -85,B 0,C 180,E1 11143.281,E2 11143.281} C_VEL
LIN {X 0,Y 409.627,Z 787.422,A -85,B 0,C 180,E1 11142.751,E2 11142.751} C_VEL
LIN {X 0,Y 401.74,Z 811.851,A -85,B 0,C 180,E1 11141.944,E2 11141.944} C_VEL
LIN {X 0,Y 392.467,Z 835.621,A -85,B 0,C 180,E1 11140.943,E2 11140.943} C_VEL
LIN {X 0,Y 383.883,Z 855.073,A -85,B 0,C 180,E1 11139.947,E2 11139.947} C_VEL
LIN {X 0,Y 372.742,Z 877.544,A -85,B 0,C 180,E1 11138.565,E2 11138.565} C_VEL
LIN {X 0,Y 361.343,Z 897.761,A -85,B 0,C 180,E1 11137.035,E2 11137.035} C_VEL
LIN {X 0,Y 350.637,Z 915.157,A -85,B 0,C 180,E1 11135.46,E2 11135.46} C_VEL
LIN {X 0,Y 337.567,Z 934.726,A -85,B 0,C 180,E1 11133.329,E2 11133.329} C_VEL
LIN {X 0,Y 324.012,Z 953.048,A -85,B 0,C 180,E1 11130.847,E2 11130.847} C_VEL
LIN {X 0,Y 312.267,Z 967.964,A -85,B 0,C 180,E1 11128.401,E2 11128.401} C_VEL
LIN {X 0,Y 297.965,Z 985.026,A -85,B 0,C 180,E1 11124.964,E2 11124.964} C_VEL
LIN {X 0,Y 285.941,Z 998.509,A -85,B 0,C 180,E1 11121.563,E2 11121.563} C_VEL
LIN {X 0,Y 274.966,Z 1010.456,A -85,B 0,C 180,E1 11117.887,E2 11117.887} C_VEL
LIN {X 0,Y 262.395,Z 1023.788,A -85,B 0,C 180,E1 11112.71,E2 11112.71} C_VEL
LIN {X 0,Y 253.792,Z 1032.921,A -85,B 0,C 180,E1 11108.21,E2 11108.21} C_VEL
LIN {X 0,Y 246.039,Z 1041.46,A -85,B 0,C 180,E1 11102.995,E2 11102.995} C_VEL
LIN {X 0,Y 239.452,Z 1049.187,A -85,B 0,C 180,E1 11096.807,E2 11096.807} C_VEL
LIN {X 0,Y 235.783,Z 1054.122,A -85,B 0,C 180,E1 11091.65,E2 11091.65} C_VEL
LIN {X 0,Y 233.463,Z 1057.949,A -85,B 0,C 180,E1 11086.389,E2 11086.389} C_VEL
LIN {X 0,Y 232.18,Z 1061.081,A -85,B 0,C 180,E1 11080.17,E2 11080.17} C_VEL
LIN {X 0,Y 231.91,Z 1062.425,A -85,B 0,C 180,E1 11074.699,E2 11074.699} C_VEL
LIN {X 0,Y 231.929,Z 1062.638,A -85,B 0,C 180,E1 11069.753,E2 11069.753} C_VEL
LIN {X 0,Y 231.913,Z 1061.92,A -85,B 0,C 180,E1 11065.053,E2 11065.053} C_VEL
LIN {X 0,Y 232.099,Z 1060.406,A -85,B 0,C 180,E1 11060.578,E2 11060.578} C_VEL
LIN {X 0,Y 232.865,Z 1057.738,A -85,B 0,C 180,E1 11055.579,E2 11055.579} C_VEL
LIN {X 0,Y 234.543,Z 1054.036,A -85,B 0,C 180,E1 11050.578,E2 11050.578} C_VEL
LIN {X 0,Y 237.719,Z 1048.756,A -85,B 0,C 180,E1 11045.127,E2 11045.127} C_VEL
LIN {X 0,Y 243.496,Z 1040.723,A -85,B 0,C 180,E1 11038.842,E2 11038.842} C_VEL
LIN {X 0,Y 249.808,Z 1032.754,A -85,B 0,C 180,E1 11033.953,E2 11033.953} C_VEL
LIN {X 0,Y 257.619,Z 1023.46,A -85,B 0,C 180,E1 11029.304,E2 11029.304} C_VEL
LIN {X 0,Y 268.837,Z 1010.267,A -85,B 0,C 180,E1 11024.068,E2 11024.068} C_VEL
LIN {X 0,Y 278.462,Z 998.845,A -85,B 0,C 180,E1 11020.427,E2 11020.427} C_VEL
LIN {X 0,Y 289.213,Z 985.822,A -85,B 0,C 180,E1 11016.982,E2 11016.982} C_VEL
LIN {X 0,Y 302.712,Z 968.635,A -85,B 0,C 180,E1 11013.313,E2 11013.313} C_VEL
LIN {X 0,Y 313.93,Z 953.506,A -85,B 0,C 180,E1 11010.688,E2 11010.688} C_VEL
LIN {X 0,Y 325.751,Z 936.62,A -85,B 0,C 180,E1 11008.244,E2 11008.244} C_VEL
LIN {X 0,Y 338.844,Z 916.191,A -85,B 0,C 180,E1 11005.84,E2 11005.84} C_VEL
LIN {X 0,Y 348.991,Z 898.956,A -85,B 0,C 180,E1 11004.164,E2 11004.164} C_VEL
LIN {X 0,Y 359.104,Z 880.276,A -85,B 0,C 180,E1 11002.628,E2 11002.628} C_VEL
LIN {X 0,Y 370.627,Z 856.425,A -85,B 0,C 180,E1 11001.022,E2 11001.022} C_VEL
LIN {X 0,Y 379.178,Z 836.342,A -85,B 0,C 180,E1 10999.913,E2 10999.913} C_VEL
LIN {X 0,Y 387.37,Z 814.664,A -85,B 0,C 180,E1 10998.924,E2 10998.924} C_VEL
LIN {X 0,Y 395.64,Z 788.671,A -85,B 0,C 180,E1 10997.979,E2 10997.979} C_VEL
LIN {X 0,Y 401.083,Z 768.126,A -85,B 0,C 180,E1 10997.386,E2 10997.386} C_VEL
LIN {X 0,Y 406.092,Z 745.116,A -85,B 0,C 180,E1 10996.855,E2 10996.855} C_VEL
LIN {X 0,Y 410.414,Z 717.437,A -85,B 0,C 180,E1 10996.352,E2 10996.352} C_VEL
LIN {X 0,Y 422.98,Z 588.251,A -85,B 0,C 180,E1 10994.403,E2 10994.403} C_VEL
LIN {X 0,Y 429.342,Z 522.138,A -85,B 0,C 180,E1 10993.399,E2 10993.399} C_VEL
LIN {X 0,Y 425.267,Z 514.206,A -85,B 0,C 180,E1 10990.568,E2 10990.568} C_VEL
LIN {X 0,Y 422.614,Z 509.372,A -85,B 0,C 180,E1 10988.298,E2 10988.298} C_VEL
LIN {X 0,Y 420.969,Z 506.231,A -85,B 0,C 180,E1 10986.547,E2 10986.547} C_VEL
LIN {X 0,Y 418.993,Z 502.394,A -85,B 0,C 180,E1 10983.694,E2 10983.694} C_VEL
LIN {X 0,Y 417.567,Z 499.574,A -85,B 0,C 180,E1 10978.353,E2 10978.353} C_VEL
LIN {X 0,Y 419.228,Z 502.687,A -85,B 0,C 180,E1 10972.738,E2 10972.738} C_VEL
LIN {X 0,Y 421.679,Z 507.537,A -85,B 0,C 180,E1 10969.48,E2 10969.48} C_VEL
LIN {X 0,Y 424.171,Z 512.251,A -85,B 0,C 180,E1 10967.129,E2 10967.129} C_VEL
LIN {X 0,Y 427.727,Z 518.934,A -85,B 0,C 180,E1 10964.475,E2 10964.475} C_VEL
LIN {X 0,Y 429.336,Z 522.331,A -85,B 0,C 180,E1 10963.412,E2 10963.412} C_VEL
LIN {X 0,Y 410.654,Z 714.446,A -85,B 0,C 180,E1 10960.538,E2 10960.538} C_VEL
LIN {X 0,Y 406.535,Z 741.359,A -85,B 0,C 180,E1 10960.051,E2 10960.051} C_VEL
LIN {X 0,Y 401.392,Z 765.218,A -85,B 0,C 180,E1 10959.493,E2 10959.493} C_VEL
LIN {X 0,Y 395.882,Z 786.235,A -85,B 0,C 180,E1 10958.862,E2 10958.862} C_VEL
LIN {X 0,Y 387.899,Z 811.521,A -85,B 0,C 180,E1 10957.923,E2 10957.923} C_VEL
LIN {X 0,Y 379.792,Z 833.093,A -85,B 0,C 180,E1 10956.926,E2 10956.926} C_VEL
LIN {X 0,Y 371.501,Z 852.652,A -85,B 0,C 180,E1 10955.84,E2 10955.84} C_VEL
LIN {X 0,Y 360.613,Z 875.496,A -85,B 0,C 180,E1 10954.308,E2 10954.308} C_VEL
LIN {X 0,Y 349.61,Z 895.876,A -85,B 0,C 180,E1 10952.627,E2 10952.627} C_VEL
LIN {X 0,Y 339.315,Z 913.363,A -85,B 0,C 180,E1 10950.907,E2 10950.907} C_VEL
LIN {X 0,Y 326.12,Z 933.868,A -85,B 0,C 180,E1 10948.468,E2 10948.468} C_VEL
LIN {X 0,Y 314.552,Z 950.339,A -85,B 0,C 180,E1 10946.063,E2 10946.063} C_VEL
LIN {X 0,Y 303.553,Z 965.105,A -85,B 0,C 180,E1 10943.487,E2 10943.487} C_VEL
LIN {X 0,Y 289.659,Z 982.654,A -85,B 0,C 180,E1 10939.718,E2 10939.718} C_VEL
LIN {X 0,Y 279.14,Z 995.291,A -85,B 0,C 180,E1 10936.35,E2 10936.35} C_VEL
LIN {X 0,Y 269.098,Z 1007.086,A -85,B 0,C 180,E1 10932.551,E2 10932.551} C_VEL
LIN {X 0,Y 258.072,Z 1019.838,A -85,B 0,C 180,E1 10927.414,E2 10927.414} C_VEL
LIN {X 0,Y 250.41,Z 1028.787,A -85,B 0,C 180,E1 10922.891,E2 10922.891} C_VEL
LIN {X 0,Y 243.575,Z 1037.222,A -85,B 0,C 180,E1 10917.637,E2 10917.637} C_VEL
LIN {X 0,Y 237.893,Z 1044.869,A -85,B 0,C 180,E1 10911.449,E2 10911.449} C_VEL
LIN {X 0,Y 234.846,Z 1049.729,A -85,B 0,C 180,E1 10906.32,E2 10906.32} C_VEL
LIN {X 0,Y 233.081,Z 1053.318,A -85,B 0,C 180,E1 10901.381,E2 10901.381} C_VEL
LIN {X 0,Y 232.181,Z 1056.025,A -85,B 0,C 180,E1 10896.18,E2 10896.18} C_VEL
LIN {X 0,Y 231.949,Z 1057.803,A -85,B 0,C 180,E1 10890.494,E2 10890.494} C_VEL
LIN {X 0,Y 231.915,Z 1058.183,A -85,B 0,C 180,E1 10885.053,E2 10885.053} C_VEL
LIN {X 0,Y 232.035,Z 1057.526,A -85,B 0,C 180,E1 10880.074,E2 10880.074} C_VEL
LIN {X 0,Y 232.573,Z 1055.887,A -85,B 0,C 180,E1 10875.051,E2 10875.051} C_VEL
LIN {X 0,Y 233.955,Z 1053.248,A -85,B 0,C 180,E1 10870.007,E2 10870.007} C_VEL
LIN {X 0,Y 236.556,Z 1049.378,A -85,B 0,C 180,E1 10864.728,E2 10864.728} C_VEL
LIN {X 0,Y 241.573,Z 1043.229,A -85,B 0,C 180,E1 10858.502,E2 10858.502} C_VEL
LIN {X 0,Y 248.298,Z 1035.648,A -85,B 0,C 180,E1 10852.84,E2 10852.84} C_VEL
LIN {X 0,Y 255.89,Z 1027.629,A -85,B 0,C 180,E1 10848.073,E2 10848.073} C_VEL
LIN {X 0,Y 267.046,Z 1016.055,A -85,B 0,C 180,E1 10842.665,E2 10842.665} C_VEL
LIN {X 0,Y 277.577,Z 1004.943,A -85,B 0,C 180,E1 10838.586,E2 10838.586} C_VEL
LIN {X 0,Y 288.374,Z 993.315,A -85,B 0,C 180,E1 10835.086,E2 10835.086} C_VEL
LIN {X 0,Y 302.699,Z 977.134,A -85,B 0,C 180,E1 10831.181,E2 10831.181} C_VEL
LIN {X 0,Y 314.78,Z 962.622,A -85,B 0,C 180,E1 10828.372,E2 10828.372} C_VEL
LIN {X 0,Y 327.55,Z 946.371,A -85,B 0,C 180,E1 10825.773,E2 10825.773} C_VEL
LIN {X 0,Y 341.372,Z 927.175,A -85,B 0,C 180,E1 10823.292,E2 10823.292} C_VEL
LIN {X 0,Y 352.498,Z 910.387,A -85,B 0,C 180,E1 10821.504,E2 10821.504} C_VEL
LIN {X 0,Y 364.018,Z 891.509,A -85,B 0,C 180,E1 10819.817,E2 10819.817} C_VEL
LIN {X 0,Y 376.241,Z 869.048,A -85,B 0,C 180,E1 10818.18,E2 10818.18} C_VEL
LIN {X 0,Y 385.323,Z 850.367,A -85,B 0,C 180,E1 10817.051,E2 10817.051} C_VEL
LIN {X 0,Y 394.24,Z 829.857,A -85,B 0,C 180,E1 10816.006,E2 10816.006} C_VEL
LIN {X 0,Y 403.954,Z 803.823,A -85,B 0,C 180,E1 10814.939,E2 10814.939} C_VEL
LIN {X 0,Y 410.588,Z 782.752,A -85,B 0,C 180,E1 10814.251,E2 10814.251} C_VEL
LIN {X 0,Y 416.262,Z 761.375,A -85,B 0,C 180,E1 10813.68,E2 10813.68} C_VEL
LIN {X 0,Y 421.956,Z 733.82,A -85,B 0,C 180,E1 10813.113,E2 10813.113} C_VEL
LIN {X 0,Y 425.262,Z 711.221,A -85,B 0,C 180,E1 10812.74,E2 10812.74} C_VEL
LIN {X 0,Y 434.982,Z 615.83,A -85,B 0,C 180,E1 10811.347,E2 10811.347} C_VEL
LIN {X 0,Y 435.52,Z 608.295,A -85,B 0,C 180,E1 10811.108,E2 10811.108} C_VEL
LIN {X 0,Y 436.213,Z 588.728,A -85,B 0,C 180,E1 10810.022,E2 10810.022} C_VEL
LIN {X 0,Y 436.738,Z 582.245,A -85,B 0,C 180,E1 10809.835,E2 10809.835} C_VEL
LIN {X 0,Y 441.233,Z 538.666,A -85,B 0,C 180,E1 10809.193,E2 10809.193} C_VEL
LIN {X 0,Y 438.554,Z 533.254,A -85,B 0,C 180,E1 10806.546,E2 10806.546} C_VEL
LIN {X 0,Y 436.916,Z 529.877,A -85,B 0,C 180,E1 10804.331,E2 10804.331} C_VEL
LIN {X 0,Y 435.354,Z 525.778,A -85,B 0,C 180,E1 10800.132,E2 10800.132} C_VEL
LIN {X 0,Y 435.424,Z 525.945,A -85,B 0,C 180,E1 10796.577,E2 10796.577} C_VEL
LIN {X 0,Y 437.389,Z 530.808,A -85,B 0,C 180,E1 10792.05,E2 10792.05} C_VEL
LIN {X 0,Y 439.316,Z 534.819,A -85,B 0,C 180,E1 10789.708,E2 10789.708} C_VEL
LIN {X 0,Y 441.287,Z 538.869,A -85,B 0,C 180,E1 10787.846,E2 10787.846} C_VEL
LIN {X 0,Y 422.779,Z 716.656,A -85,B 0,C 180,E1 10785.298,E2 10785.298} C_VEL
LIN {X 0,Y 418.437,Z 743.583,A -85,B 0,C 180,E1 10784.848,E2 10784.848} C_VEL
LIN {X 0,Y 413.096,Z 767.161,A -85,B 0,C 180,E1 10784.359,E2 10784.359} C_VEL
LIN {X 0,Y 407.544,Z 787.21,A -85,B 0,C 180,E1 10783.847,E2 10783.847} C_VEL
LIN {X 0,Y 399.76,Z 811.075,A -85,B 0,C 180,E1 10783.08,E2 10783.08} C_VEL
LIN {X 0,Y 390.501,Z 834.583,A -85,B 0,C 180,E1 10782.121,E2 10782.121} C_VEL
LIN {X 0,Y 381.903,Z 853.846,A -85,B 0,C 180,E1 10781.168,E2 10781.168} C_VEL
LIN {X 0,Y 371.037,Z 875.594,A -85,B 0,C 180,E1 10779.88,E2 10779.88} C_VEL
LIN {X 0,Y 358.96,Z 896.779,A -85,B 0,C 180,E1 10778.329,E2 10778.329} C_VEL
LIN {X 0,Y 347.72,Z 914.721,A -85,B 0,C 180,E1 10776.742,E2 10776.742} C_VEL
LIN {X 0,Y 334.211,Z 934.534,A -85,B 0,C 180,E1 10774.624,E2 10774.624} C_VEL
LIN {X 0,Y 320.816,Z 952.237,A -85,B 0,C 180,E1 10772.269,E2 10772.269} C_VEL
LIN {X 0,Y 308.721,Z 967.215,A -85,B 0,C 180,E1 10769.855,E2 10769.855} C_VEL
LIN {X 0,Y 294.59,Z 983.693,A -85,B 0,C 180,E1 10766.612,E2 10766.612} C_VEL
LIN {X 0,Y 281.45,Z 997.926,A -85,B 0,C 180,E1 10763.067,E2 10763.067} C_VEL
LIN {X 0,Y 270.542,Z 1009.348,A -85,B 0,C 180,E1 10759.583,E2 10759.583} C_VEL
LIN {X 0,Y 258.244,Z 1021.965,A -85,B 0,C 180,E1 10754.804,E2 10754.804} C_VEL
LIN {X 0,Y 248.098,Z 1032.111,A -85,B 0,C 180,E1 10749.852,E2 10749.852} C_VEL
LIN {X 0,Y 240.303,Z 1040.158,A -85,B 0,C 180,E1 10744.944,E2 10744.944} C_VEL
LIN {X 0,Y 232.794,Z 1048.391,A -85,B 0,C 180,E1 10738.474,E2 10738.474} C_VEL
LIN {X 0,Y 228.304,Z 1053.874,A -85,B 0,C 180,E1 10732.669,E2 10732.669} C_VEL
LIN {X 0,Y 225.734,Z 1057.721,A -85,B 0,C 180,E1 10727.264,E2 10727.264} C_VEL
LIN {X 0,Y 224.304,Z 1060.713,A -85,B 0,C 180,E1 10721.272,E2 10721.272} C_VEL
LIN {X 0,Y 223.923,Z 1062.28,A -85,B 0,C 180,E1 10715.638,E2 10715.638} C_VEL
LIN {X 0,Y 223.927,Z 1062.601,A -85,B 0,C 180,E1 10710.256,E2 10710.256} C_VEL
LIN {X 0,Y 223.91,Z 1061.967,A -85,B 0,C 180,E1 10705.39,E2 10705.39} C_VEL
LIN {X 0,Y 224.11,Z 1060.38,A -85,B 0,C 180,E1 10700.408,E2 10700.408} C_VEL
LIN {X 0,Y 224.977,Z 1057.628,A -85,B 0,C 180,E1 10695.062,E2 10695.062} C_VEL
LIN {X 0,Y 226.808,Z 1053.916,A -85,B 0,C 180,E1 10689.888,E2 10689.888} C_VEL
LIN {X 0,Y 230.245,Z 1048.625,A -85,B 0,C 180,E1 10684.261,E2 10684.261} C_VEL
LIN {X 0,Y 236.472,Z 1040.493,A -85,B 0,C 180,E1 10677.745,E2 10677.745} C_VEL
LIN {X 0,Y 243.112,Z 1032.598,A -85,B 0,C 180,E1 10672.801,E2 10672.801} C_VEL
LIN {X 0,Y 251.336,Z 1023.285,A -85,B 0,C 180,E1 10668.06,E2 10668.06} C_VEL
LIN {X 0,Y 262.999,Z 1010.176,A -85,B 0,C 180,E1 10662.798,E2 10662.798} C_VEL
LIN {X 0,Y 273.119,Z 998.635,A -85,B 0,C 180,E1 10659.093,E2 10659.093} C_VEL
LIN {X 0,Y 284.847,Z 984.927,A -85,B 0,C 180,E1 10655.474,E2 10655.474} C_VEL
LIN {X 0,Y 298.215,Z 968.38,A -85,B 0,C 180,E1 10651.975,E2 10651.975} C_VEL
LIN {X 0,Y 309.766,Z 953.235,A -85,B 0,C 180,E1 10649.364,E2 10649.364} C_VEL
LIN {X 0,Y 322.274,Z 935.819,A -85,B 0,C 180,E1 10646.875,E2 10646.875} C_VEL
LIN {X 0,Y 335.323,Z 915.859,A -85,B 0,C 180,E1 10644.569,E2 10644.569} C_VEL
LIN {X 0,Y 345.921,Z 898.217,A -85,B 0,C 180,E1 10642.884,E2 10642.884} C_VEL
LIN {X 0,Y 356.99,Z 878.118,A -85,B 0,C 180,E1 10641.277,E2 10641.277} C_VEL
LIN {X 0,Y 367.772,Z 855.976,A -85,B 0,C 180,E1 10639.832,E2 10639.832} C_VEL
LIN {X 0,Y 376.455,Z 835.901,A -85,B 0,C 180,E1 10638.747,E2 10638.747} C_VEL
LIN {X 0,Y 385.247,Z 812.925,A -85,B 0,C 180,E1 10637.726,E2 10637.726} C_VEL
LIN {X 0,Y 393.216,Z 787.949,A -85,B 0,C 180,E1 10636.851,E2 10636.851} C_VEL
LIN {X 0,Y 398.691,Z 767.528,A -85,B 0,C 180,E1 10636.28,E2 10636.28} C_VEL
LIN {X 0,Y 403.933,Z 743.637,A -85,B 0,C 180,E1 10635.745,E2 10635.745} C_VEL
LIN {X 0,Y 408.096,Z 716.812,A -85,B 0,C 180,E1 10635.27,E2 10635.27} C_VEL
LIN {X 0,Y 426.827,Z 527.76,A -85,B 0,C 180,E1 10632.463,E2 10632.463} C_VEL
LIN {X 0,Y 423.178,Z 520.582,A -85,B 0,C 180,E1 10629.726,E2 10629.726} C_VEL
LIN {X 0,Y 421.206,Z 516.81,A -85,B 0,C 180,E1 10627.914,E2 10627.914} C_VEL
LIN {X 0,Y 419.751,Z 513.942,A -85,B 0,C 180,E1 10626.291,E2 10626.291} C_VEL
LIN {X 0,Y 417.936,Z 510.279,A -85,B 0,C 180,E1 10623.566,E2 10623.566} C_VEL
LIN {X 0,Y 416.591,Z 507.519,A -85,B 0,C 180,E1 10618.35,E2 10618.35} C_VEL
LIN {X 0,Y 418.165,Z 510.609,A -85,B 0,C 180,E1 10612.857,E2 10612.857} C_VEL
LIN {X 0,Y 420.503,Z 515.368,A -85,B 0,C 180,E1 10609.658,E2 10609.658} C_VEL
LIN {X 0,Y 422.785,Z 519.802,A -85,B 0,C 180,E1 10607.433,E2 10607.433} C_VEL
LIN {X 0,Y 426.236,Z 526.5,A -85,B 0,C 180,E1 10604.767,E2 10604.767} C_VEL
LIN {X 0,Y 426.785,Z 527.877,A -85,B 0,C 180,E1 10604.372,E2 10604.372} C_VEL
LIN {X 0,Y 408.259,Z 714.569,A -85,B 0,C 180,E1 10601.608,E2 10601.608} C_VEL
LIN {X 0,Y 404.052,Z 741.58,A -85,B 0,C 180,E1 10601.127,E2 10601.127} C_VEL
LIN {X 0,Y 398.87,Z 765.263,A -85,B 0,C 180,E1 10600.585,E2 10600.585} C_VEL
LIN {X 0,Y 393.406,Z 785.817,A -85,B 0,C 180,E1 10599.982,E2 10599.982} C_VEL
LIN {X 0,Y 385.794,Z 809.864,A -85,B 0,C 180,E1 10599.12,E2 10599.12} C_VEL
LIN {X 0,Y 377.171,Z 832.527,A -85,B 0,C 180,E1 10598.102,E2 10598.102} C_VEL
LIN {X 0,Y 368.65,Z 852.333,A -85,B 0,C 180,E1 10597.026,E2 10597.026} C_VEL
LIN {X 0,Y 357.592,Z 875.177,A -85,B 0,C 180,E1 10595.526,E2 10595.526} C_VEL
LIN {X 0,Y 346.357,Z 895.595,A -85,B 0,C 180,E1 10593.872,E2 10593.872} C_VEL
LIN {X 0,Y 336.167,Z 912.563,A -85,B 0,C 180,E1 10592.236,E2 10592.236} C_VEL
LIN {X 0,Y 323.383,Z 932.175,A -85,B 0,C 180,E1 10589.968,E2 10589.968} C_VEL
LIN {X 0,Y 310.762,Z 949.716,A -85,B 0,C 180,E1 10587.457,E2 10587.457} C_VEL
LIN {X 0,Y 299.799,Z 964.05,A -85,B 0,C 180,E1 10584.994,E2 10584.994} C_VEL
LIN {X 0,Y 286.863,Z 980.125,A -85,B 0,C 180,E1 10581.652,E2 10581.652} C_VEL
LIN {X 0,Y 274.557,Z 994.378,A -85,B 0,C 180,E1 10577.925,E2 10577.925} C_VEL
LIN {X 0,Y 264.611,Z 1005.603,A -85,B 0,C 180,E1 10574.351,E2 10574.351} C_VEL
LIN {X 0,Y 253.825,Z 1017.666,A -85,B 0,C 180,E1 10569.655,E2 10569.655} C_VEL
LIN {X 0,Y 244.281,Z 1028.163,A -85,B 0,C 180,E1 10564.392,E2 10564.392} C_VEL
LIN {X 0,Y 237.491,Z 1035.993,A -85,B 0,C 180,E1 10559.511,E2 10559.511} C_VEL
LIN {X 0,Y 231.322,Z 1043.755,A -85,B 0,C 180,E1 10553.432,E2 10553.432} C_VEL
LIN {X 0,Y 227.27,Z 1049.525,A -85,B 0,C 180,E1 10547.309,E2 10547.309} C_VEL
LIN {X 0,Y 225.237,Z 1053.276,A -85,B 0,C 180,E1 10542.043,E2 10542.043} C_VEL
LIN {X 0,Y 224.256,Z 1055.905,A -85,B 0,C 180,E1 10536.914,E2 10536.914} C_VEL
LIN {X 0,Y 223.946,Z 1057.492,A -85,B 0,C 180,E1 10532.047,E2 10532.047} C_VEL
LIN {X 0,Y 223.906,Z 1058.156,A -85,B 0,C 180,E1 10527.697,E2 10527.697} C_VEL
LIN {X 0,Y 223.943,Z 1058.123,A -85,B 0,C 180,E1 10523.334,E2 10523.334} C_VEL
LIN {X 0,Y 224.126,Z 1057.321,A -85,B 0,C 180,E1 10518.679,E2 10518.679} C_VEL
LIN {X 0,Y 224.836,Z 1055.602,A -85,B 0,C 180,E1 10513.729,E2 10513.729} C_VEL
LIN {X 0,Y 226.628,Z 1052.656,A -85,B 0,C 180,E1 10508.247,E2 10508.247} C_VEL
LIN {X 0,Y 230.919,Z 1047.169,A -85,B 0,C 180,E1 10501.273,E2 10501.273} C_VEL
LIN {X 0,Y 236.291,Z 1041.186,A -85,B 0,C 180,E1 10495.75,E2 10495.75} C_VEL
LIN {X 0,Y 243.125,Z 1034.159,A -85,B 0,C 180,E1 10490.641,E2 10490.641} C_VEL
LIN {X 0,Y 253.589,Z 1023.758,A -85,B 0,C 180,E1 10484.787,E2 10484.787} C_VEL
LIN {X 0,Y 263.737,Z 1013.63,A -85,B 0,C 180,E1 10480.356,E2 10480.356} C_VEL
LIN {X 0,Y 274.892,Z 1002.36,A -85,B 0,C 180,E1 10476.363,E2 10476.363} C_VEL
LIN {X 0,Y 288.998,Z 987.47,A -85,B 0,C 180,E1 10472.196,E2 10472.196} C_VEL
LIN {X 0,Y 300.754,Z 974.382,A -85,B 0,C 180,E1 10469.257,E2 10469.257} C_VEL
LIN {X 0,Y 313.76,Z 959.102,A -85,B 0,C 180,E1 10466.429,E2 10466.429} C_VEL
LIN {X 0,Y 327.985,Z 940.98,A -85,B 0,C 180,E1 10463.729,E2 10463.729} C_VEL
LIN {X 0,Y 339.518,Z 925.066,A -85,B 0,C 180,E1 10461.782,E2 10461.782} C_VEL
LIN {X 0,Y 351.428,Z 907.306,A -85,B 0,C 180,E1 10459.964,E2 10459.964} C_VEL
LIN {X 0,Y 364.995,Z 884.819,A -85,B 0,C 180,E1 10458.087,E2 10458.087} C_VEL
LIN {X 0,Y 375.43,Z 865.484,A -85,B 0,C 180,E1 10456.773,E2 10456.773} C_VEL
LIN {X 0,Y 385.629,Z 844.456,A -85,B 0,C 180,E1 10455.581,E2 10455.581} C_VEL
LIN {X 0,Y 395.536,Z 820.793,A -85,B 0,C 180,E1 10454.489,E2 10454.489} C_VEL
LIN {X 0,Y 402.94,Z 800.332,A -85,B 0,C 180,E1 10453.712,E2 10453.712} C_VEL
LIN {X 0,Y 409.982,Z 777.681,A -85,B 0,C 180,E1 10453.013,E2 10453.013} C_VEL
LIN {X 0,Y 416.582,Z 751.133,A -85,B 0,C 180,E1 10452.383,E2 10452.383} C_VEL
LIN {X 0,Y 420.768,Z 729.288,A -85,B 0,C 180,E1 10451.976,E2 10451.976} C_VEL
LIN {X 0,Y 424.315,Z 703.498,A -85,B 0,C 180,E1 10451.57,E2 10451.57} C_VEL
LIN {X 0,Y 436.738,Z 582.245,A -85,B 0,C 180,E1 10449.835,E2 10449.835} C_VEL
LIN {X 0,Y 437.328,Z 574.71,A -85,B 0,C 180,E1 10449.602,E2 10449.602} C_VEL
LIN {X 0,Y 438.226,Z 555.16,A -85,B 0,C 180,E1 10448.517,E2 10448.517} C_VEL
LIN {X 0,Y 438.784,Z 548.679,A -85,B 0,C 180,E1 10448.33,E2 10448.33} C_VEL
LIN {X 0,Y 439.165,Z 544.733,A -85,B 0,C 180,E1 10448.247,E2 10448.247} C_VEL
LIN {X 0,Y 437.228,Z 540.76,A -85,B 0,C 180,E1 10446.17,E2 10446.17} C_VEL
LIN {X 0,Y 435.766,Z 537.647,A -85,B 0,C 180,E1 10444.079,E2 10444.079} C_VEL
LIN {X 0,Y 434.354,Z 533.701,A -85,B 0,C 180,E1 10440,E2 10440} C_VEL
LIN {X 0,Y 434.437,Z 533.988,A -85,B 0,C 180,E1 10436.569,E2 10436.569} C_VEL
LIN {X 0,Y 436.313,Z 538.73,A -85,B 0,C 180,E1 10432.163,E2 10432.163} C_VEL
LIN {X 0,Y 438.139,Z 542.655,A -85,B 0,C 180,E1 10429.879,E2 10429.879} C_VEL
LIN {X 0,Y 439.208,Z 545.008,A -85,B 0,C 180,E1 10428.788,E2 10428.788} C_VEL
LIN {X 0,Y 421.011,Z 716.604,A -85,B 0,C 180,E1 10426.362,E2 10426.362} C_VEL
LIN {X 0,Y 416.594,Z 743.585,A -85,B 0,C 180,E1 10425.92,E2 10425.92} C_VEL
LIN {X 0,Y 411.212,Z 767.043,A -85,B 0,C 180,E1 10425.446,E2 10425.446} C_VEL
LIN {X 0,Y 405.394,Z 787.739,A -85,B 0,C 180,E1 10424.932,E2 10424.932} C_VEL
LIN {X 0,Y 397.063,Z 812.616,A -85,B 0,C 180,E1 10424.144,E2 10424.144} C_VEL
LIN {X 0,Y 387.733,Z 835.781,A -85,B 0,C 180,E1 10423.212,E2 10423.212} C_VEL
LIN {X 0,Y 378.951,Z 855.03,A -85,B 0,C 180,E1 10422.273,E2 10422.273} C_VEL
LIN {X 0,Y 367.131,Z 877.989,A -85,B 0,C 180,E1 10420.919,E2 10420.919} C_VEL
LIN {X 0,Y 355.524,Z 897.808,A -85,B 0,C 180,E1 10419.478,E2 10419.478} C_VEL
LIN {X 0,Y 344.182,Z 915.496,A -85,B 0,C 180,E1 10417.93,E2 10417.93} C_VEL
LIN {X 0,Y 329.709,Z 936.06,A -85,B 0,C 180,E1 10415.736,E2 10415.736} C_VEL
LIN {X 0,Y 316.329,Z 953.268,A -85,B 0,C 180,E1 10413.449,E2 10413.449} C_VEL
LIN {X 0,Y 303.952,Z 968.15,A -85,B 0,C 180,E1 10411.05,E2 10411.05} C_VEL
LIN {X 0,Y 288.776,Z 985.152,A -85,B 0,C 180,E1 10407.656,E2 10407.656} C_VEL
LIN {X 0,Y 275.922,Z 998.608,A -85,B 0,C 180,E1 10404.265,E2 10404.265} C_VEL
LIN {X 0,Y 264.095,Z 1010.529,A -85,B 0,C 180,E1 10400.566,E2 10400.566} C_VEL
LIN {X 0,Y 250.719,Z 1023.537,A -85,B 0,C 180,E1 10395.42,E2 10395.42} C_VEL
LIN {X 0,Y 241.345,Z 1032.518,A -85,B 0,C 180,E1 10390.888,E2 10390.888} C_VEL
LIN {X 0,Y 232.627,Z 1041.088,A -85,B 0,C 180,E1 10385.469,E2 10385.469} C_VEL
LIN {X 0,Y 224.983,Z 1048.945,A -85,B 0,C 180,E1 10378.892,E2 10378.892} C_VEL
LIN {X 0,Y 220.558,Z 1054.043,A -85,B 0,C 180,E1 10373.229,E2 10373.229} C_VEL
LIN {X 0,Y 217.741,Z 1057.995,A -85,B 0,C 180,E1 10367.367,E2 10367.367} C_VEL
LIN {X 0,Y 216.227,Z 1061.02,A -85,B 0,C 180,E1 10360.659,E2 10360.659} C_VEL
LIN {X 0,Y 215.913,Z 1062.277,A -85,B 0,C 180,E1 10355.048,E2 10355.048} C_VEL
LIN {X 0,Y 215.938,Z 1062.496,A -85,B 0,C 180,E1 10350,E2 10350} C_VEL
LIN {X 0,Y 215.915,Z 1061.807,A -85,B 0,C 180,E1 10344.952,E2 10344.952} C_VEL
LIN {X 0,Y 216.157,Z 1060.204,A -85,B 0,C 180,E1 10339.876,E2 10339.876} C_VEL
LIN {X 0,Y 217.102,Z 1057.517,A -85,B 0,C 180,E1 10334.507,E2 10334.507} C_VEL
LIN {X 0,Y 219.107,Z 1053.795,A -85,B 0,C 180,E1 10329.149,E2 10329.149} C_VEL
LIN {X 0,Y 223.029,Z 1048.236,A -85,B 0,C 180,E1 10323.076,E2 10323.076} C_VEL
LIN {X 0,Y 229.406,Z 1040.419,A -85,B 0,C 180,E1 10316.689,E2 10316.689} C_VEL
LIN {X 0,Y 236.525,Z 1032.434,A -85,B 0,C 180,E1 10311.58,E2 10311.58} C_VEL
LIN {X 0,Y 245.629,Z 1022.645,A -85,B 0,C 180,E1 10306.532,E2 10306.532} C_VEL
LIN {X 0,Y 257.394,Z 1009.978,A -85,B 0,C 180,E1 10301.433,E2 10301.433} C_VEL
LIN {X 0,Y 267.928,Z 998.422,A -85,B 0,C 180,E1 10297.706,E2 10297.706} C_VEL
LIN {X 0,Y 280.083,Z 984.701,A -85,B 0,C 180,E1 10294.083,E2 10294.083} C_VEL
LIN {X 0,Y 293.888,Z 968.125,A -85,B 0,C 180,E1 10290.597,E2 10290.597} C_VEL
LIN {X 0,Y 305.775,Z 952.963,A -85,B 0,C 180,E1 10288.006,E2 10288.006} C_VEL
LIN {X 0,Y 318.989,Z 935.015,A -85,B 0,C 180,E1 10285.479,E2 10285.479} C_VEL
LIN {X 0,Y 332.343,Z 914.939,A -85,B 0,C 180,E1 10283.212,E2 10283.212} C_VEL
LIN {X 0,Y 343.013,Z 897.502,A -85,B 0,C 180,E1 10281.583,E2 10281.583} C_VEL
LIN {X 0,Y 354.919,Z 876.216,A -85,B 0,C 180,E1 10279.931,E2 10279.931} C_VEL
LIN {X 0,Y 365.495,Z 854.616,A -85,B 0,C 180,E1 10278.573,E2 10278.573} C_VEL
LIN {X 0,Y 373.89,Z 835.46,A -85,B 0,C 180,E1 10277.565,E2 10277.565} C_VEL
LIN {X 0,Y 382.847,Z 812.379,A -85,B 0,C 180,E1 10276.565,E2 10276.565} C_VEL
LIN {X 0,Y 390.633,Z 788.315,A -85,B 0,C 180,E1 10275.743,E2 10275.743} C_VEL
LIN {X 0,Y 396.249,Z 767.72,A -85,B 0,C 180,E1 10275.18,E2 10275.18} C_VEL
LIN {X 0,Y 401.454,Z 744.409,A -85,B 0,C 180,E1 10274.668,E2 10274.668} C_VEL
LIN {X 0,Y 405.82,Z 717.056,A -85,B 0,C 180,E1 10274.19,E2 10274.19} C_VEL
LIN {X 0,Y 421.065,Z 566.3,A -85,B 0,C 180,E1 10271.973,E2 10271.973} C_VEL
LIN {X 0,Y 424.377,Z 533.321,A -85,B 0,C 180,E1 10271.484,E2 10271.484} C_VEL
LIN {X 0,Y 421.261,Z 527.047,A -85,B 0,C 180,E1 10268.944,E2 10268.944} C_VEL
LIN {X 0,Y 418.653,Z 521.823,A -85,B 0,C 180,E1 10266.17,E2 10266.17} C_VEL
LIN {X 0,Y 416.88,Z 518.163,A -85,B 0,C 180,E1 10263.438,E2 10263.438} C_VEL
LIN {X 0,Y 415.616,Z 515.464,A -85,B 0,C 180,E1 10258.346,E2 10258.346} C_VEL
LIN {X 0,Y 417.133,Z 518.623,A -85,B 0,C 180,E1 10252.919,E2 10252.919} C_VEL
LIN {X 0,Y 419.332,Z 523.199,A -85,B 0,C 180,E1 10249.837,E2 10249.837} C_VEL
LIN {X 0,Y 421.56,Z 527.662,A -85,B 0,C 180,E1 10247.605,E2 10247.605} C_VEL
LIN {X 0,Y 424.355,Z 533.407,A -85,B 0,C 180,E1 10245.342,E2 10245.342} C_VEL
LIN {X 0,Y 406.014,Z 714.649,A -85,B 0,C 180,E1 10242.69,E2 10242.69} C_VEL
LIN {X 0,Y 401.74,Z 741.668,A -85,B 0,C 180,E1 10242.219,E2 10242.219} C_VEL
LIN {X 0,Y 396.473,Z 765.397,A -85,B 0,C 180,E1 10241.687,E2 10241.687} C_VEL
LIN {X 0,Y 390.836,Z 786.25,A -85,B 0,C 180,E1 10241.089,E2 10241.089} C_VEL
LIN {X 0,Y 382.598,Z 811.561,A -85,B 0,C 180,E1 10240.19,E2 10240.19} C_VEL
LIN {X 0,Y 374.259,Z 833.051,A -85,B 0,C 180,E1 10239.24,E2 10239.24} C_VEL
LIN {X 0,Y 365.227,Z 853.614,A -85,B 0,C 180,E1 10238.138,E2 10238.138} C_VEL
LIN {X 0,Y 353.129,Z 877.767,A -85,B 0,C 180,E1 10236.549,E2 10236.549} C_VEL
LIN {X 0,Y 342.489,Z 896.635,A -85,B 0,C 180,E1 10235.025,E2 10235.025} C_VEL
LIN {X 0,Y 331.338,Z 914.721,A -85,B 0,C 180,E1 10233.284,E2 10233.284} C_VEL
LIN {X 0,Y 317.198,Z 935.489,A -85,B 0,C 180,E1 10230.829,E2 10230.829} C_VEL
LIN {X 0,Y 305.759,Z 950.922,A -85,B 0,C 180,E1 10228.596,E2 10228.596} C_VEL
LIN {X 0,Y 294.133,Z 965.653,A -85,B 0,C 180,E1 10226.043,E2 10226.043} C_VEL
LIN {X 0,Y 279.247,Z 983.271,A -85,B 0,C 180,E1 10222.244,E2 10222.244} C_VEL
LIN {X 0,Y 268.096,Z 995.745,A -85,B 0,C 180,E1 10218.883,E2 10218.883} C_VEL
LIN {X 0,Y 256.238,Z 1008.645,A -85,B 0,C 180,E1 10214.619,E2 10214.619} C_VEL
LIN {X 0,Y 244.891,Z 1020.58,A -85,B 0,C 180,E1 10209.564,E2 10209.564} C_VEL
LIN {X 0,Y 236.447,Z 1029.535,A -85,B 0,C 180,E1 10204.812,E2 10204.812} C_VEL
LIN {X 0,Y 228.358,Z 1038.562,A -85,B 0,C 180,E1 10198.793,E2 10198.793} C_VEL
LIN {X 0,Y 222.608,Z 1045.397,A -85,B 0,C 180,E1 10192.723,E2 10192.723} C_VEL
LIN {X 0,Y 219.188,Z 1050.187,A -85,B 0,C 180,E1 10187.248,E2 10187.248} C_VEL
LIN {X 0,Y 217.074,Z 1054.021,A -85,B 0,C 180,E1 10181.424,E2 10181.424} C_VEL
LIN {X 0,Y 216.075,Z 1056.913,A -85,B 0,C 180,E1 10174.778,E2 10174.778} C_VEL
LIN {X 0,Y 215.921,Z 1058.103,A -85,B 0,C 180,E1 10169.204,E2 10169.204} C_VEL
LIN {X 0,Y 215.93,Z 1058.284,A -85,B 0,C 180,E1 10164.153,E2 10164.153} C_VEL
LIN {X 0,Y 216.099,Z 1057.585,A -85,B 0,C 180,E1 10159.064,E2 10159.064} C_VEL
LIN {X 0,Y 216.841,Z 1055.88,A -85,B 0,C 180,E1 10153.663,E2 10153.663} C_VEL
LIN {X 0,Y 218.603,Z 1053.147,A -85,B 0,C 180,E1 10148.206,E2 10148.206} C_VEL
LIN {X 0,Y 222.358,Z 1048.618,A -85,B 0,C 180,E1 10141.826,E2 10141.826} C_VEL
LIN {X 0,Y 228.497,Z 1042.104,A -85,B 0,C 180,E1 10135.328,E2 10135.328} C_VEL
LIN {X 0,Y 235.46,Z 1035.288,A -85,B 0,C 180,E1 10130.117,E2 10130.117} C_VEL
LIN {X 0,Y 244.931,Z 1026.38,A -85,B 0,C 180,E1 10124.739,E2 10124.739} C_VEL
LIN {X 0,Y 256.744,Z 1015.139,A -85,B 0,C 180,E1 10119.546,E2 10119.546} C_VEL
LIN {X 0,Y 267.741,Z 1004.468,A -85,B 0,C 180,E1 10115.633,E2 10115.633} C_VEL
LIN {X 0,Y 281.605,Z 990.612,A -85,B 0,C 180,E1 10111.553,E2 10111.553} C_VEL
LIN {X 0,Y 295.749,Z 975.383,A -85,B 0,C 180,E1 10108.066,E2 10108.066} C_VEL
LIN {X 0,Y 307.911,Z 961.538,A -85,B 0,C 180,E1 10105.478,E2 10105.478} C_VEL
LIN {X 0,Y 322.57,Z 943.675,A -85,B 0,C 180,E1 10102.754,E2 10102.754} C_VEL
LIN {X 0,Y 335.906,Z 925.756,A -85,B 0,C 180,E1 10100.564,E2 10100.564} C_VEL
LIN {X 0,Y 347.582,Z 908.76,A -85,B 0,C 180,E1 10098.839,E2 10098.839} C_VEL
LIN {X 0,Y 361.344,Z 886.641,A -85,B 0,C 180,E1 10096.998,E2 10096.998} C_VEL
LIN {X 0,Y 372.285,Z 866.831,A -85,B 0,C 180,E1 10095.664,E2 10095.664} C_VEL
LIN {X 0,Y 381.813,Z 847.669,A -85,B 0,C 180,E1 10094.586,E2 10094.586} C_VEL
LIN {X 0,Y 392.253,Z 823.783,A -85,B 0,C 180,E1 10093.475,E2 10093.475} C_VEL
LIN {X 0,Y 400.385,Z 801.882,A -85,B 0,C 180,E1 10092.65,E2 10092.65} C_VEL
LIN {X 0,Y 407.11,Z 780.836,A -85,B 0,C 180,E1 10092.006,E2 10092.006} C_VEL
LIN {X 0,Y 413.787,Z 755.611,A -85,B 0,C 180,E1 10091.397,E2 10091.397} C_VEL
LIN {X 0,Y 418.627,Z 731.334,A -85,B 0,C 180,E1 10090.943,E2 10090.943} C_VEL
LIN {X 0,Y 421.903,Z 708.836,A -85,B 0,C 180,E1 10090.59,E2 10090.59} C_VEL
LIN {X 0,Y 438.784,Z 548.679,A -85,B 0,C 180,E1 10088.33,E2 10088.33} C_VEL
LIN {X 0,Y 438.802,Z 546.773,A -85,B 0,C 180,E1 10088.163,E2 10088.163} C_VEL
LIN {X 0,Y 438.448,Z 545.622,A -85,B 0,C 180,E1 10087.774,E2 10087.774} C_VEL
LIN {X 0,Y 437.657,Z 545.679,A -85,B 0,C 180,E1 10087.123,E2 10087.123} C_VEL
LIN {X 0,Y 435.904,Z 547.651,A -85,B 0,C 180,E1 10085.696,E2 10085.696} C_VEL
LIN {X 0,Y 435.495,Z 547.37,A -85,B 0,C 180,E1 10085.219,E2 10085.219} C_VEL
LIN {X 0,Y 434.705,Z 545.523,A -85,B 0,C 180,E1 10083.957,E2 10083.957} C_VEL
LIN {X 0,Y 433.378,Z 541.642,A -85,B 0,C 180,E1 10080,E2 10080} C_VEL
LIN {X 0,Y 433.437,Z 541.873,A -85,B 0,C 180,E1 10076.694,E2 10076.694} C_VEL
LIN {X 0,Y 435.197,Z 546.539,A -85,B 0,C 180,E1 10072.342,E2 10072.342} C_VEL
LIN {X 0,Y 436.966,Z 550.488,A -85,B 0,C 180,E1 10070.051,E2 10070.051} C_VEL
LIN {X 0,Y 437.23,Z 551.321,A -85,B 0,C 180,E1 10069.737,E2 10069.737} C_VEL
LIN {X 0,Y 419.375,Z 716.657,A -85,B 0,C 180,E1 10067.433,E2 10067.433} C_VEL
LIN {X 0,Y 414.842,Z 743.845,A -85,B 0,C 180,E1 10066.996,E2 10066.996} C_VEL
LIN {X 0,Y 409.449,Z 767.032,A -85,B 0,C 180,E1 10066.541,E2 10066.541} C_VEL
LIN {X 0,Y 403.612,Z 787.536,A -85,B 0,C 180,E1 10066.048,E2 10066.048} C_VEL
LIN {X 0,Y 395.394,Z 811.881,A -85,B 0,C 180,E1 10065.302,E2 10065.302} C_VEL
LIN {X 0,Y 386.147,Z 834.623,A -85,B 0,C 180,E1 10064.419,E2 10064.419} C_VEL
LIN {X 0,Y 377.413,Z 853.582,A -85,B 0,C 180,E1 10063.532,E2 10063.532} C_VEL
LIN {X 0,Y 365.84,Z 875.993,A -85,B 0,C 180,E1 10062.268,E2 10062.268} C_VEL
LIN {X 0,Y 353.175,Z 897.34,A -85,B 0,C 180,E1 10060.766,E2 10060.766} C_VEL
LIN {X 0,Y 341.659,Z 914.995,A -85,B 0,C 180,E1 10059.261,E2 10059.261} C_VEL
LIN {X 0,Y 327.531,Z 934.794,A -85,B 0,C 180,E1 10057.212,E2 10057.212} C_VEL
LIN {X 0,Y 313.208,Z 952.821,A -85,B 0,C 180,E1 10054.875,E2 10054.875} C_VEL
LIN {X 0,Y 300.782,Z 967.403,A -85,B 0,C 180,E1 10052.571,E2 10052.571} C_VEL
LIN {X 0,Y 285.82,Z 983.82,A -85,B 0,C 180,E1 10049.382,E2 10049.382} C_VEL
LIN {X 0,Y 271.801,Z 998.025,A -85,B 0,C 180,E1 10045.865,E2 10045.865} C_VEL
LIN {X 0,Y 259.479,Z 1009.993,A -85,B 0,C 180,E1 10042.181,E2 10042.181} C_VEL
LIN {X 0,Y 245.156,Z 1023.367,A -85,B 0,C 180,E1 10036.892,E2 10036.892} C_VEL
LIN {X 0,Y 235.119,Z 1032.52,A -85,B 0,C 180,E1 10032.216,E2 10032.216} C_VEL
LIN {X 0,Y 225.909,Z 1041.078,A -85,B 0,C 180,E1 10026.692,E2 10026.692} C_VEL
LIN {X 0,Y 217.847,Z 1048.843,A -85,B 0,C 180,E1 10020.02,E2 10020.02} C_VEL
LIN {X 0,Y 213.011,Z 1054.004,A -85,B 0,C 180,E1 10014.103,E2 10014.103} C_VEL
LIN {X 0,Y 209.945,Z 1057.947,A -85,B 0,C 180,E1 10008.033,E2 10008.033} C_VEL
LIN {X 0,Y 208.27,Z 1060.954,A -85,B 0,C 180,E1 10001.072,E2 10001.072} C_VEL
LIN {X 0,Y 207.916,Z 1062.203,A -85,B 0,C 180,E1 9995.243,E2 9995.243} C_VEL
LIN {X 0,Y 207.938,Z 1062.414,A -85,B 0,C 180,E1 9990,E2 9990} C_VEL
LIN {X 0,Y 207.913,Z 1061.784,A -85,B 0,C 180,E1 9985.034,E2 9985.034} C_VEL
LIN {X 0,Y 208.165,Z 1060.219,A -85,B 0,C 180,E1 9979.763,E2 9979.763} C_VEL
LIN {X 0,Y 209.168,Z 1057.568,A -85,B 0,C 180,E1 9974.188,E2 9974.188} C_VEL
LIN {X 0,Y 211.3,Z 1053.884,A -85,B 0,C 180,E1 9968.631,E2 9968.631} C_VEL
LIN {X 0,Y 215.233,Z 1048.621,A -85,B 0,C 180,E1 9962.619,E2 9962.619} C_VEL
LIN {X 0,Y 222.497,Z 1040.266,A -85,B 0,C 180,E1 9955.512,E2 9955.512} C_VEL
LIN {X 0,Y 230.046,Z 1032.271,A -85,B 0,C 180,E1 9950.288,E2 9950.288} C_VEL
LIN {X 0,Y 239.633,Z 1022.47,A -85,B 0,C 180,E1 9945.158,E2 9945.158} C_VEL
LIN {X 0,Y 251.938,Z 1009.778,A -85,B 0,C 180,E1 9940.007,E2 9940.007} C_VEL
LIN {X 0,Y 262.898,Z 998.21,A -85,B 0,C 180,E1 9936.264,E2 9936.264} C_VEL
LIN {X 0,Y 276.148,Z 983.766,A -85,B 0,C 180,E1 9932.472,E2 9932.472} C_VEL
LIN {X 0,Y 290.292,Z 967.195,A -85,B 0,C 180,E1 9929.056,E2 9929.056} C_VEL
LIN {X 0,Y 301.963,Z 952.689,A -85,B 0,C 180,E1 9926.614,E2 9926.614} C_VEL
LIN {X 0,Y 315.899,Z 934.196,A -85,B 0,C 180,E1 9924.054,E2 9924.054} C_VEL
LIN {X 0,Y 329.194,Z 914.58,A -85,B 0,C 180,E1 9921.888,E2 9921.888} C_VEL
LIN {X 0,Y 340.069,Z 897.145,A -85,B 0,C 180,E1 9920.292,E2 9920.292} C_VEL
LIN {X 0,Y 352.453,Z 875.309,A -85,B 0,C 180,E1 9918.642,E2 9918.642} C_VEL
LIN {X 0,Y 362.973,Z 854.164,A -85,B 0,C 180,E1 9917.349,E2 9917.349} C_VEL
LIN {X 0,Y 371.511,Z 834.964,A -85,B 0,C 180,E1 9916.366,E2 9916.366} C_VEL
LIN {X 0,Y 380.667,Z 811.672,A -85,B 0,C 180,E1 9915.385,E2 9915.385} C_VEL
LIN {X 0,Y 388.485,Z 787.696,A -85,B 0,C 180,E1 9914.591,E2 9914.591} C_VEL
LIN {X 0,Y 394.144,Z 767.171,A -85,B 0,C 180,E1 9914.049,E2 9914.049} C_VEL
LIN {X 0,Y 399.584,Z 742.988,A -85,B 0,C 180,E1 9913.536,E2 9913.536} C_VEL
LIN {X 0,Y 403.81,Z 716.314,A -85,B 0,C 180,E1 9913.083,E2 9913.083} C_VEL
LIN {X 0,Y 422.052,Z 539.084,A -85,B 0,C 180,E1 9910.511,E2 9910.511} C_VEL
LIN {X 0,Y 419.084,Z 532.901,A -85,B 0,C 180,E1 9907.816,E2 9907.816} C_VEL
LIN {X 0,Y 417.338,Z 529.36,A -85,B 0,C 180,E1 9905.775,E2 9905.775} C_VEL
LIN {X 0,Y 415.827,Z 526.048,A -85,B 0,C 180,E1 9903.308,E2 9903.308} C_VEL
LIN {X 0,Y 414.64,Z 523.409,A -85,B 0,C 180,E1 9898.342,E2 9898.342} C_VEL
LIN {X 0,Y 416.078,Z 526.556,A -85,B 0,C 180,E1 9893.029,E2 9893.029} C_VEL
LIN {X 0,Y 418.108,Z 530.894,A -85,B 0,C 180,E1 9890.085,E2 9890.085} C_VEL
LIN {X 0,Y 420.265,Z 535.366,A -85,B 0,C 180,E1 9887.845,E2 9887.845} C_VEL
LIN {X 0,Y 422.018,Z 539.228,A -85,B 0,C 180,E1 9886.32,E2 9886.32} C_VEL
LIN {X 0,Y 403.909,Z 714.777,A -85,B 0,C 180,E1 9883.784,E2 9883.784} C_VEL
LIN {X 0,Y 399.561,Z 741.827,A -85,B 0,C 180,E1 9883.322,E2 9883.322} C_VEL
LIN {X 0,Y 394.222,Z 765.541,A -85,B 0,C 180,E1 9882.803,E2 9882.803} C_VEL
LIN {X 0,Y 388.513,Z 786.344,A -85,B 0,C 180,E1 9882.22,E2 9882.22} C_VEL
LIN {X 0,Y 380.39,Z 811.019,A -85,B 0,C 180,E1 9881.37,E2 9881.37} C_VEL
LIN {X 0,Y 371.916,Z 832.58,A -85,B 0,C 180,E1 9880.443,E2 9880.443} C_VEL
LIN {X 0,Y 363.146,Z 852.31,A -85,B 0,C 180,E1 9879.415,E2 9879.415} C_VEL
LIN {X 0,Y 352.051,Z 874.537,A -85,B 0,C 180,E1 9878.02,E2 9878.02} C_VEL
LIN {X 0,Y 340.355,Z 895.033,A -85,B 0,C 180,E1 9876.431,E2 9876.431} C_VEL
LIN {X 0,Y 329.752,Z 912.008,A -85,B 0,C 180,E1 9874.86,E2 9874.86} C_VEL
LIN {X 0,Y 316.319,Z 931.786,A -85,B 0,C 180,E1 9872.653,E2 9872.653} C_VEL
LIN {X 0,Y 303.034,Z 949.382,A -85,B 0,C 180,E1 9870.202,E2 9870.202} C_VEL
LIN {X 0,Y 291.023,Z 964.256,A -85,B 0,C 180,E1 9867.693,E2 9867.693} C_VEL
LIN {X 0,Y 277.01,Z 980.61,A -85,B 0,C 180,E1 9864.306,E2 9864.306} C_VEL
LIN {X 0,Y 263.971,Z 994.717,A -85,B 0,C 180,E1 9860.599,E2 9860.599} C_VEL
LIN {X 0,Y 252.828,Z 1006.361,A -85,B 0,C 180,E1 9856.828,E2 9856.828} C_VEL
LIN {X 0,Y 240.473,Z 1018.958,A -85,B 0,C 180,E1 9851.703,E2 9851.703} C_VEL
LIN {X 0,Y 230.946,Z 1028.511,A -85,B 0,C 180,E1 9846.689,E2 9846.689} C_VEL
LIN {X 0,Y 223.389,Z 1036.317,A -85,B 0,C 180,E1 9841.58,E2 9841.58} C_VEL
LIN {X 0,Y 216.221,Z 1044.283,A -85,B 0,C 180,E1 9834.886,E2 9834.886} C_VEL
LIN {X 0,Y 211.88,Z 1049.704,A -85,B 0,C 180,E1 9828.717,E2 9828.717} C_VEL
LIN {X 0,Y 209.556,Z 1053.35,A -85,B 0,C 180,E1 9823.24,E2 9823.24} C_VEL
LIN {X 0,Y 208.351,Z 1056.002,A -85,B 0,C 180,E1 9817.722,E2 9817.722} C_VEL
LIN {X 0,Y 207.958,Z 1057.611,A -85,B 0,C 180,E1 9812.48,E2 9812.48} C_VEL
LIN {X 0,Y 207.909,Z 1058.277,A -85,B 0,C 180,E1 9808.071,E2 9808.071} C_VEL
LIN {X 0,Y 207.943,Z 1058.313,A -85,B 0,C 180,E1 9803.373,E2 9803.373} C_VEL
LIN {X 0,Y 208.151,Z 1057.581,A -85,B 0,C 180,E1 9798.36,E2 9798.36} C_VEL
LIN {X 0,Y 209.046,Z 1055.821,A -85,B 0,C 180,E1 9792.749,E2 9792.749} C_VEL
LIN {X 0,Y 211.179,Z 1052.899,A -85,B 0,C 180,E1 9786.86,E2 9786.86} C_VEL
LIN {X 0,Y 215.922,Z 1047.718,A -85,B 0,C 180,E1 9779.685,E2 9779.685} C_VEL
LIN {X 0,Y 222.272,Z 1041.507,A -85,B 0,C 180,E1 9773.573,E2 9773.573} C_VEL
LIN {X 0,Y 229.839,Z 1034.579,A -85,B 0,C 180,E1 9768.271,E2 9768.271} C_VEL
LIN {X 0,Y 240.997,Z 1024.624,A -85,B 0,C 180,E1 9762.395,E2 9762.395} C_VEL
LIN {X 0,Y 252.56,Z 1014.065,A -85,B 0,C 180,E1 9757.646,E2 9757.646} C_VEL
LIN {X 0,Y 264.375,Z 1003.052,A -85,B 0,C 180,E1 9753.689,E2 9753.689} C_VEL
LIN {X 0,Y 279.997,Z 987.716,A -85,B 0,C 180,E1 9749.386,E2 9749.386} C_VEL
LIN {X 0,Y 292.616,Z 974.509,A -85,B 0,C 180,E1 9746.457,E2 9746.457} C_VEL
LIN {X 0,Y 305.921,Z 959.721,A -85,B 0,C 180,E1 9743.771,E2 9743.771} C_VEL
LIN {X 0,Y 321.409,Z 940.969,A -85,B 0,C 180,E1 9741.048,E2 9741.048} C_VEL
LIN {X 0,Y 333.457,Z 925.067,A -85,B 0,C 180,E1 9739.171,E2 9739.171} C_VEL
LIN {X 0,Y 345.836,Z 907.337,A -85,B 0,C 180,E1 9737.427,E2 9737.427} C_VEL
LIN {X 0,Y 359.872,Z 884.908,A -85,B 0,C 180,E1 9735.635,E2 9735.635} C_VEL
LIN {X 0,Y 370.584,Z 865.724,A -85,B 0,C 180,E1 9734.39,E2 9734.39} C_VEL
LIN {X 0,Y 381.111,Z 844.71,A -85,B 0,C 180,E1 9733.256,E2 9733.256} C_VEL
LIN {X 0,Y 391.279,Z 821.192,A -85,B 0,C 180,E1 9732.225,E2 9732.225} C_VEL
LIN {X 0,Y 398.942,Z 800.64,A -85,B 0,C 180,E1 9731.485,E2 9731.485} C_VEL
LIN {X 0,Y 406.176,Z 778.017,A -85,B 0,C 180,E1 9730.821,E2 9730.821} C_VEL
LIN {X 0,Y 413.007,Z 751.285,A -85,B 0,C 180,E1 9730.221,E2 9730.221} C_VEL
LIN {X 0,Y 417.332,Z 729.276,A -85,B 0,C 180,E1 9729.832,E2 9729.832} C_VEL
LIN {X 0,Y 420.999,Z 703.324,A -85,B 0,C 180,E1 9729.439,E2 9729.439} C_VEL
LIN {X 0,Y 437.226,Z 551.059,A -85,B 0,C 180,E1 9727.325,E2 9727.325} C_VEL
LIN {X 0,Y 435.921,Z 548.262,A -85,B 0,C 180,E1 9725.792,E2 9725.792} C_VEL
LIN {X 0,Y 435.495,Z 547.37,A -85,B 0,C 180,E1 9725.219,E2 9725.219} C_VEL
LIN {X 0,Y 435.008,Z 547.283,A -85,B 0,C 180,E1 9724.635,E2 9724.635} C_VEL
LIN {X 0,Y 433.94,Z 549.643,A -85,B 0,C 180,E1 9723.587,E2 9723.587} C_VEL
LIN {X 0,Y 433.095,Z 551.764,A -85,B 0,C 180,E1 9722.623,E2 9722.623} C_VEL
LIN {X 0,Y 432.837,Z 551.81,A -85,B 0,C 180,E1 9722.126,E2 9722.126} C_VEL
LIN {X 0,Y 432.38,Z 549.567,A -85,B 0,C 180,E1 9719.868,E2 9719.868} C_VEL
LIN {X 0,Y 432.438,Z 549.758,A -85,B 0,C 180,E1 9716.819,E2 9716.819} C_VEL
LIN {X 0,Y 434.125,Z 554.46,A -85,B 0,C 180,E1 9712.456,E2 9712.456} C_VEL
LIN {X 0,Y 435.407,Z 557.316,A -85,B 0,C 180,E1 9710.699,E2 9710.699} C_VEL
LIN {X 0,Y 417.901,Z 716.605,A -85,B 0,C 180,E1 9708.513,E2 9708.513} C_VEL
LIN {X 0,Y 413.294,Z 743.847,A -85,B 0,C 180,E1 9708.086,E2 9708.086} C_VEL
LIN {X 0,Y 407.837,Z 767.021,A -85,B 0,C 180,E1 9707.645,E2 9707.645} C_VEL
LIN {X 0,Y 401.76,Z 788.067,A -85,B 0,C 180,E1 9707.154,E2 9707.154} C_VEL
LIN {X 0,Y 392.986,Z 813.392,A -85,B 0,C 180,E1 9706.393,E2 9706.393} C_VEL
LIN {X 0,Y 384.066,Z 834.96,A -85,B 0,C 180,E1 9705.574,E2 9705.574} C_VEL
LIN {X 0,Y 375.039,Z 854.22,A -85,B 0,C 180,E1 9704.696,E2 9704.696} C_VEL
LIN {X 0,Y 363.023,Z 876.977,A -85,B 0,C 180,E1 9703.437,E2 9703.437} C_VEL
LIN {X 0,Y 350.583,Z 897.537,A -85,B 0,C 180,E1 9702.02,E2 9702.02} C_VEL
LIN {X 0,Y 338.771,Z 915.294,A -85,B 0,C 180,E1 9700.537,E2 9700.537} C_VEL
LIN {X 0,Y 324.45,Z 934.924,A -85,B 0,C 180,E1 9698.544,E2 9698.544} C_VEL
LIN {X 0,Y 310.12,Z 952.57,A -85,B 0,C 180,E1 9696.301,E2 9696.301} C_VEL
LIN {X 0,Y 297.814,Z 966.673,A -85,B 0,C 180,E1 9694.121,E2 9694.121} C_VEL
LIN {X 0,Y 283.129,Z 982.444,A -85,B 0,C 180,E1 9691.143,E2 9691.143} C_VEL
LIN {X 0,Y 267.736,Z 997.602,A -85,B 0,C 180,E1 9687.467,E2 9687.467} C_VEL
LIN {X 0,Y 255.698,Z 1008.888,A -85,B 0,C 180,E1 9684.043,E2 9684.043} C_VEL
LIN {X 0,Y 242.255,Z 1021.08,A -85,B 0,C 180,E1 9679.415,E2 9679.415} C_VEL
LIN {X 0,Y 229.965,Z 1031.712,A -85,B 0,C 180,E1 9674.081,E2 9674.081} C_VEL
LIN {X 0,Y 220.835,Z 1039.655,A -85,B 0,C 180,E1 9669.003,E2 9669.003} C_VEL
LIN {X 0,Y 212.111,Z 1047.578,A -85,B 0,C 180,E1 9662.455,E2 9662.455} C_VEL
LIN {X 0,Y 205.91,Z 1053.55,A -85,B 0,C 180,E1 9655.606,E2 9655.606} C_VEL
LIN {X 0,Y 202.527,Z 1057.416,A -85,B 0,C 180,E1 9649.616,E2 9649.616} C_VEL
LIN {X 0,Y 200.605,Z 1060.296,A -85,B 0,C 180,E1 9643.255,E2 9643.255} C_VEL
LIN {X 0,Y 199.955,Z 1062.035,A -85,B 0,C 180,E1 9636.604,E2 9636.604} C_VEL
LIN {X 0,Y 199.917,Z 1062.399,A -85,B 0,C 180,E1 9630.86,E2 9630.86} C_VEL
LIN {X 0,Y 199.91,Z 1061.831,A -85,B 0,C 180,E1 9625.41,E2 9625.41} C_VEL
LIN {X 0,Y 200.174,Z 1060.233,A -85,B 0,C 180,E1 9619.641,E2 9619.641} C_VEL
LIN {X 0,Y 201.325,Z 1057.457,A -85,B 0,C 180,E1 9613.555,E2 9613.555} C_VEL
LIN {X 0,Y 203.663,Z 1053.762,A -85,B 0,C 180,E1 9607.788,E2 9607.788} C_VEL
LIN {X 0,Y 207.912,Z 1048.489,A -85,B 0,C 180,E1 9601.569,E2 9601.569} C_VEL
LIN {X 0,Y 215.687,Z 1040.114,A -85,B 0,C 180,E1 9594.26,E2 9594.26} C_VEL
LIN {X 0,Y 223.684,Z 1032.106,A -85,B 0,C 180,E1 9588.921,E2 9588.921} C_VEL
LIN {X 0,Y 234.289,Z 1021.829,A -85,B 0,C 180,E1 9583.489,E2 9583.489} C_VEL
LIN {X 0,Y 246.644,Z 1009.578,A -85,B 0,C 180,E1 9578.518,E2 9578.518} C_VEL
LIN {X 0,Y 258.328,Z 997.701,A -85,B 0,C 180,E1 9574.68,E2 9574.68} C_VEL
LIN {X 0,Y 272.44,Z 982.805,A -85,B 0,C 180,E1 9570.818,E2 9570.818} C_VEL
LIN {X 0,Y 286.499,Z 966.756,A -85,B 0,C 180,E1 9567.568,E2 9567.568} C_VEL
LIN {X 0,Y 298.335,Z 952.416,A -85,B 0,C 180,E1 9565.188,E2 9565.188} C_VEL
LIN {X 0,Y 312.639,Z 933.857,A -85,B 0,C 180,E1 9562.665,E2 9562.665} C_VEL
LIN {X 0,Y 326.165,Z 914.308,A -85,B 0,C 180,E1 9560.549,E2 9560.549} C_VEL
LIN {X 0,Y 337.301,Z 896.786,A -85,B 0,C 180,E1 9558.98,E2 9558.98} C_VEL
LIN {X 0,Y 349.915,Z 874.892,A -85,B 0,C 180,E1 9557.368,E2 9557.368} C_VEL
LIN {X 0,Y 360.491,Z 853.981,A -85,B 0,C 180,E1 9556.124,E2 9556.124} C_VEL
LIN {X 0,Y 368.858,Z 835.485,A -85,B 0,C 180,E1 9555.198,E2 9555.198} C_VEL
LIN {X 0,Y 378.23,Z 812.055,A -85,B 0,C 180,E1 9554.232,E2 9554.232} C_VEL
LIN {X 0,Y 386.216,Z 788.017,A -85,B 0,C 180,E1 9553.455,E2 9553.455} C_VEL
LIN {X 0,Y 392.028,Z 767.257,A -85,B 0,C 180,E1 9552.921,E2 9552.921} C_VEL
LIN {X 0,Y 397.457,Z 743.486,A -85,B 0,C 180,E1 9552.429,E2 9552.429} C_VEL
LIN {X 0,Y 401.83,Z 716.535,A -85,B 0,C 180,E1 9551.979,E2 9551.979} C_VEL
LIN {X 0,Y 419.85,Z 544.857,A -85,B 0,C 180,E1 9549.527,E2 9549.527} C_VEL
LIN {X 0,Y 417.513,Z 539.979,A -85,B 0,C 180,E1 9547.223,E2 9547.223} C_VEL
LIN {X 0,Y 416.145,Z 537.068,A -85,B 0,C 180,E1 9545.515,E2 9545.515} C_VEL
LIN {X 0,Y 414.704,Z 533.852,A -85,B 0,C 180,E1 9543.041,E2 9543.041} C_VEL
LIN {X 0,Y 413.664,Z 531.354,A -85,B 0,C 180,E1 9538.338,E2 9538.338} C_VEL
LIN {X 0,Y 414.988,Z 534.363,A -85,B 0,C 180,E1 9533.22,E2 9533.22} C_VEL
LIN {X 0,Y 416.933,Z 538.69,A -85,B 0,C 180,E1 9530.283,E2 9530.283} C_VEL
LIN {X 0,Y 418.983,Z 543.08,A -85,B 0,C 180,E1 9528.082,E2 9528.082} C_VEL
LIN {X 0,Y 419.804,Z 545.042,A -85,B 0,C 180,E1 9527.309,E2 9527.309} C_VEL
LIN {X 0,Y 401.947,Z 714.929,A -85,B 0,C 180,E1 9524.889,E2 9524.889} C_VEL
LIN {X 0,Y 397.532,Z 741.971,A -85,B 0,C 180,E1 9524.436,E2 9524.436} C_VEL
LIN {X 0,Y 392.151,Z 765.56,A -85,B 0,C 180,E1 9523.933,E2 9523.933} C_VEL
LIN {X 0,Y 386.371,Z 786.337,A -85,B 0,C 180,E1 9523.368,E2 9523.368} C_VEL
LIN {X 0,Y 377.913,Z 811.596,A -85,B 0,C 180,E1 9522.518,E2 9522.518} C_VEL
LIN {X 0,Y 369.312,Z 833.103,A -85,B 0,C 180,E1 9521.613,E2 9521.613} C_VEL
LIN {X 0,Y 360.405,Z 852.788,A -85,B 0,C 180,E1 9520.609,E2 9520.609} C_VEL
LIN {X 0,Y 348.702,Z 875.67,A -85,B 0,C 180,E1 9519.193,E2 9519.193} C_VEL
LIN {X 0,Y 337.209,Z 895.409,A -85,B 0,C 180,E1 9517.688,E2 9517.688} C_VEL
LIN {X 0,Y 326.431,Z 912.307,A -85,B 0,C 180,E1 9516.151,E2 9516.151} C_VEL
LIN {X 0,Y 312.672,Z 932.099,A -85,B 0,C 180,E1 9513.975,E2 9513.975} C_VEL
LIN {X 0,Y 299.07,Z 949.671,A -85,B 0,C 180,E1 9511.557,E2 9511.557} C_VEL
LIN {X 0,Y 286.746,Z 964.528,A -85,B 0,C 180,E1 9509.071,E2 9509.071} C_VEL
LIN {X 0,Y 272.319,Z 980.85,A -85,B 0,C 180,E1 9505.704,E2 9505.704} C_VEL
LIN {X 0,Y 258.851,Z 994.944,A -85,B 0,C 180,E1 9501.999,E2 9501.999} C_VEL
LIN {X 0,Y 247.624,Z 1006.24,A -85,B 0,C 180,E1 9498.332,E2 9498.332} C_VEL
LIN {X 0,Y 234.906,Z 1018.691,A -85,B 0,C 180,E1 9493.259,E2 9493.259} C_VEL
LIN {X 0,Y 224.428,Z 1028.685,A -85,B 0,C 180,E1 9487.939,E2 9487.939} C_VEL
LIN {X 0,Y 216.12,Z 1036.827,A -85,B 0,C 180,E1 9482.458,E2 9482.458} C_VEL
LIN {X 0,Y 208.367,Z 1044.922,A -85,B 0,C 180,E1 9475.282,E2 9475.282} C_VEL
LIN {X 0,Y 204.047,Z 1050.034,A -85,B 0,C 180,E1 9469.167,E2 9469.167} C_VEL
LIN {X 0,Y 201.518,Z 1053.78,A -85,B 0,C 180,E1 9463.193,E2 9463.193} C_VEL
LIN {X 0,Y 200.247,Z 1056.554,A -85,B 0,C 180,E1 9456.883,E2 9456.883} C_VEL
LIN {X 0,Y 199.95,Z 1058.157,A -85,B 0,C 180,E1 9450.573,E2 9450.573} C_VEL
LIN {X 0,Y 199.919,Z 1058.519,A -85,B 0,C 180,E1 9444.835,E2 9444.835} C_VEL
LIN {X 0,Y 200.098,Z 1057.912,A -85,B 0,C 180,E1 9439.054,E2 9439.054} C_VEL
LIN {X 0,Y 200.987,Z 1056.211,A -85,B 0,C 180,E1 9432.931,E2 9432.931} C_VEL
LIN {X 0,Y 203.013,Z 1053.564,A -85,B 0,C 180,E1 9427.077,E2 9427.077} C_VEL
LIN {X 0,Y 206.645,Z 1049.711,A -85,B 0,C 180,E1 9421.062,E2 9421.062} C_VEL
LIN {X 0,Y 213.261,Z 1043.636,A -85,B 0,C 180,E1 9414.121,E2 9414.121} C_VEL
LIN {X 0,Y 221.948,Z 1035.991,A -85,B 0,C 180,E1 9407.836,E2 9407.836} C_VEL
LIN {X 0,Y 231.373,Z 1027.975,A -85,B 0,C 180,E1 9402.721,E2 9402.721} C_VEL
LIN {X 0,Y 244.611,Z 1016.609,A -85,B 0,C 180,E1 9397.147,E2 9397.147} C_VEL
LIN {X 0,Y 257.238,Z 1005.302,A -85,B 0,C 180,E1 9392.903,E2 9392.903} C_VEL
LIN {X 0,Y 270.411,Z 993.042,A -85,B 0,C 180,E1 9389.233,E2 9389.233} C_VEL
LIN {X 0,Y 286.026,Z 977.511,A -85,B 0,C 180,E1 9385.589,E2 9385.589} C_VEL
LIN {X 0,Y 298.781,Z 963.859,A -85,B 0,C 180,E1 9383.03,E2 9383.03} C_VEL
LIN {X 0,Y 311.514,Z 949.29,A -85,B 0,C 180,E1 9380.774,E2 9380.774} C_VEL
LIN {X 0,Y 327.055,Z 929.978,A -85,B 0,C 180,E1 9378.355,E2 9378.355} C_VEL
LIN {X 0,Y 340.048,Z 912.042,A -85,B 0,C 180,E1 9376.549,E2 9376.549} C_VEL
LIN {X 0,Y 351.475,Z 894.823,A -85,B 0,C 180,E1 9375.107,E2 9375.107} C_VEL
LIN {X 0,Y 364.233,Z 873.625,A -85,B 0,C 180,E1 9373.641,E2 9373.641} C_VEL
LIN {X 0,Y 375.237,Z 852.679,A -85,B 0,C 180,E1 9372.465,E2 9372.465} C_VEL
LIN {X 0,Y 384.243,Z 833.448,A -85,B 0,C 180,E1 9371.559,E2 9371.559} C_VEL
LIN {X 0,Y 394.092,Z 809.55,A -85,B 0,C 180,E1 9370.637,E2 9370.637} C_VEL
LIN {X 0,Y 402.232,Z 785.581,A -85,B 0,C 180,E1 9369.911,E2 9369.911} C_VEL
LIN {X 0,Y 408.078,Z 765.137,A -85,B 0,C 180,E1 9369.409,E2 9369.409} C_VEL
LIN {X 0,Y 413.956,Z 739.913,A -85,B 0,C 180,E1 9368.918,E2 9368.918} C_VEL
LIN {X 0,Y 418.195,Z 713.807,A -85,B 0,C 180,E1 9368.513,E2 9368.513} C_VEL
LIN {X 0,Y 435.389,Z 557.223,A -85,B 0,C 180,E1 9366.365,E2 9366.365} C_VEL
LIN {X 0,Y 433.646,Z 553.4,A -85,B 0,C 180,E1 9363.834,E2 9363.834} C_VEL
LIN {X 0,Y 432.837,Z 551.81,A -85,B 0,C 180,E1 9362.126,E2 9362.126} C_VEL
LIN {X 0,Y 432.448,Z 551.793,A -85,B 0,C 180,E1 9361.172,E2 9361.172} C_VEL
LIN {X 0,Y 431.765,Z 554.288,A -85,B 0,C 180,E1 9359.65,E2 9359.65} C_VEL
LIN {X 0,Y 431.345,Z 557.226,A -85,B 0,C 180,E1 9357.968,E2 9357.968} C_VEL
LIN {X 0,Y 431.366,Z 557.523,A -85,B 0,C 180,E1 9357.445,E2 9357.445} C_VEL
LIN {X 0,Y 431.499,Z 558.249,A -85,B 0,C 180,E1 9356.413,E2 9356.413} C_VEL
LIN {X 0,Y 433.016,Z 562.268,A -85,B 0,C 180,E1 9352.637,E2 9352.637} C_VEL
LIN {X 0,Y 433.633,Z 564.008,A -85,B 0,C 180,E1 9351.66,E2 9351.66} C_VEL
LIN {X 0,Y 416.577,Z 716.553,A -85,B 0,C 180,E1 9349.601,E2 9349.601} C_VEL
LIN {X 0,Y 411.897,Z 743.849,A -85,B 0,C 180,E1 9349.183,E2 9349.183} C_VEL
LIN {X 0,Y 406.406,Z 766.903,A -85,B 0,C 180,E1 9348.759,E2 9348.759} C_VEL
LIN {X 0,Y 400.288,Z 787.863,A -85,B 0,C 180,E1 9348.288,E2 9348.288} C_VEL
LIN {X 0,Y 391.634,Z 812.658,A -85,B 0,C 180,E1 9347.571,E2 9347.571} C_VEL
LIN {X 0,Y 382.144,Z 835.297,A -85,B 0,C 180,E1 9346.741,E2 9346.741} C_VEL
LIN {X 0,Y 373.186,Z 854.123,A -85,B 0,C 180,E1 9345.91,E2 9345.91} C_VEL
LIN {X 0,Y 360.799,Z 877.204,A -85,B 0,C 180,E1 9344.669,E2 9344.669} C_VEL
LIN {X 0,Y 348.205,Z 897.67,A -85,B 0,C 180,E1 9343.296,E2 9343.296} C_VEL
LIN {X 0,Y 336.187,Z 915.408,A -85,B 0,C 180,E1 9341.852,E2 9341.852} C_VEL
LIN {X 0,Y 321.134,Z 935.558,A -85,B 0,C 180,E1 9339.843,E2 9339.843} C_VEL
LIN {X 0,Y 306.912,Z 952.682,A -85,B 0,C 180,E1 9337.704,E2 9337.704} C_VEL
LIN {X 0,Y 293.752,Z 967.378,A -85,B 0,C 180,E1 9335.463,E2 9335.463} C_VEL
LIN {X 0,Y 277.763,Z 983.95,A -85,B 0,C 180,E1 9332.319,E2 9332.319} C_VEL
LIN {X 0,Y 262.855,Z 998.127,A -85,B 0,C 180,E1 9328.858,E2 9328.858} C_VEL
LIN {X 0,Y 249.634,Z 1010.069,A -85,B 0,C 180,E1 9325.196,E2 9325.196} C_VEL
LIN {X 0,Y 234.086,Z 1023.394,A -85,B 0,C 180,E1 9319.87,E2 9319.87} C_VEL
LIN {X 0,Y 223.075,Z 1032.524,A -85,B 0,C 180,E1 9315.089,E2 9315.089} C_VEL
LIN {X 0,Y 212.4,Z 1041.415,A -85,B 0,C 180,E1 9309.11,E2 9309.11} C_VEL
LIN {X 0,Y 203.661,Z 1048.785,A -85,B 0,C 180,E1 9302.354,E2 9302.354} C_VEL
LIN {X 0,Y 198.284,Z 1053.719,A -85,B 0,C 180,E1 9296.344,E2 9296.344} C_VEL
LIN {X 0,Y 194.586,Z 1057.658,A -85,B 0,C 180,E1 9289.888,E2 9289.888} C_VEL
LIN {X 0,Y 192.43,Z 1060.754,A -85,B 0,C 180,E1 9282.301,E2 9282.301} C_VEL
LIN {X 0,Y 191.931,Z 1062.032,A -85,B 0,C 180,E1 9275.981,E2 9275.981} C_VEL
LIN {X 0,Y 191.927,Z 1062.272,A -85,B 0,C 180,E1 9270.299,E2 9270.299} C_VEL
LIN {X 0,Y 191.914,Z 1061.67,A -85,B 0,C 180,E1 9264.919,E2 9264.919} C_VEL
LIN {X 0,Y 192.215,Z 1060.132,A -85,B 0,C 180,E1 9259.207,E2 9259.207} C_VEL
LIN {X 0,Y 193.478,Z 1057.392,A -85,B 0,C 180,E1 9252.956,E2 9252.956} C_VEL
LIN {X 0,Y 196.067,Z 1053.641,A -85,B 0,C 180,E1 9246.879,E2 9246.879} C_VEL
LIN {X 0,Y 200.92,Z 1048.098,A -85,B 0,C 180,E1 9240.155,E2 9240.155} C_VEL
LIN {X 0,Y 208.989,Z 1039.96,A -85,B 0,C 180,E1 9232.927,E2 9232.927} C_VEL
LIN {X 0,Y 217.455,Z 1031.941,A -85,B 0,C 180,E1 9227.474,E2 9227.474} C_VEL
LIN {X 0,Y 228.623,Z 1021.653,A -85,B 0,C 180,E1 9221.97,E2 9221.97} C_VEL
LIN {X 0,Y 241.521,Z 1009.377,A -85,B 0,C 180,E1 9216.964,E2 9216.964} C_VEL
LIN {X 0,Y 253.367,Z 997.783,A -85,B 0,C 180,E1 9213.214,E2 9213.214} C_VEL
LIN {X 0,Y 267.562,Z 983.312,A -85,B 0,C 180,E1 9209.457,E2 9209.457} C_VEL
LIN {X 0,Y 282.003,Z 967.355,A -85,B 0,C 180,E1 9206.227,E2 9206.227} C_VEL
LIN {X 0,Y 294.194,Z 952.995,A -85,B 0,C 180,E1 9203.857,E2 9203.857} C_VEL
LIN {X 0,Y 308.314,Z 935.166,A -85,B 0,C 180,E1 9201.446,E2 9201.446} C_VEL
LIN {X 0,Y 322.163,Z 915.757,A -85,B 0,C 180,E1 9199.35,E2 9199.35} C_VEL
LIN {X 0,Y 333.869,Z 897.778,A -85,B 0,C 180,E1 9197.757,E2 9197.757} C_VEL
LIN {X 0,Y 346.263,Z 876.872,A -85,B 0,C 180,E1 9196.232,E2 9196.232} C_VEL
LIN {X 0,Y 357.998,Z 854.166,A -85,B 0,C 180,E1 9194.901,E2 9194.901} C_VEL
LIN {X 0,Y 366.805,Z 834.985,A -85,B 0,C 180,E1 9193.969,E2 9193.969} C_VEL
LIN {X 0,Y 376.165,Z 811.876,A -85,B 0,C 180,E1 9193.046,E2 9193.046} C_VEL
LIN {X 0,Y 384.487,Z 787.05,A -85,B 0,C 180,E1 9192.269,E2 9192.269} C_VEL
LIN {X 0,Y 390.334,Z 766.309,A -85,B 0,C 180,E1 9191.759,E2 9191.759} C_VEL
LIN {X 0,Y 396.165,Z 740.765,A -85,B 0,C 180,E1 9191.253,E2 9191.253} C_VEL
LIN {X 0,Y 400.229,Z 714.939,A -85,B 0,C 180,E1 9190.838,E2 9190.838} C_VEL
LIN {X 0,Y 417.742,Z 550.881,A -85,B 0,C 180,E1 9188.534,E2 9188.534} C_VEL
LIN {X 0,Y 415.421,Z 545.575,A -85,B 0,C 180,E1 9185.871,E2 9185.871} C_VEL
LIN {X 0,Y 413.657,Z 541.736,A -85,B 0,C 180,E1 9182.91,E2 9182.91} C_VEL
LIN {X 0,Y 412.688,Z 539.299,A -85,B 0,C 180,E1 9178.334,E2 9178.334} C_VEL
LIN {X 0,Y 413.933,Z 542.278,A -85,B 0,C 180,E1 9173.342,E2 9173.342} C_VEL
LIN {X 0,Y 415.736,Z 546.418,A -85,B 0,C 180,E1 9170.517,E2 9170.517} C_VEL
LIN {X 0,Y 417.719,Z 550.817,A -85,B 0,C 180,E1 9168.31,E2 9168.31} C_VEL
LIN {X 0,Y 400.145,Z 715.008,A -85,B 0,C 180,E1 9166.005,E2 9166.005} C_VEL
LIN {X 0,Y 395.641,Z 742.179,A -85,B 0,C 180,E1 9165.56,E2 9165.56} C_VEL
LIN {X 0,Y 390.189,Z 765.757,A -85,B 0,C 180,E1 9165.071,E2 9165.071} C_VEL
LIN {X 0,Y 384.386,Z 786.326,A -85,B 0,C 180,E1 9164.528,E2 9164.528} C_VEL
LIN {X 0,Y 376.028,Z 811.048,A -85,B 0,C 180,E1 9163.724,E2 9163.724} C_VEL
LIN {X 0,Y 366.866,Z 833.621,A -85,B 0,C 180,E1 9162.8,E2 9162.8} C_VEL
LIN {X 0,Y 357.822,Z 853.263,A -85,B 0,C 180,E1 9161.82,E2 9161.82} C_VEL
LIN {X 0,Y 345.926,Z 876.075,A -85,B 0,C 180,E1 9160.439,E2 9160.439} C_VEL
LIN {X 0,Y 334.121,Z 895.957,A -85,B 0,C 180,E1 9158.954,E2 9158.954} C_VEL
LIN {X 0,Y 322.765,Z 913.372,A -85,B 0,C 180,E1 9157.393,E2 9157.393} C_VEL
LIN {X 0,Y 308.122,Z 933.774,A -85,B 0,C 180,E1 9155.154,E2 9155.154} C_VEL
LIN {X 0,Y 294.524,Z 950.875,A -85,B 0,C 180,E1 9152.806,E2 9152.806} C_VEL
LIN {X 0,Y 281.915,Z 965.635,A -85,B 0,C 180,E1 9150.337,E2 9150.337} C_VEL
LIN {X 0,Y 265.746,Z 983.165,A -85,B 0,C 180,E1 9146.645,E2 9146.645} C_VEL
LIN {X 0,Y 253.254,Z 995.795,A -85,B 0,C 180,E1 9143.271,E2 9143.271} C_VEL
LIN {X 0,Y 241.065,Z 1007.603,A -85,B 0,C 180,E1 9139.367,E2 9139.367} C_VEL
LIN {X 0,Y 227.465,Z 1020.234,A -85,B 0,C 180,E1 9133.99,E2 9133.99} C_VEL
LIN {X 0,Y 217.585,Z 1029.257,A -85,B 0,C 180,E1 9129.018,E2 9129.018} C_VEL
LIN {X 0,Y 208.555,Z 1037.684,A -85,B 0,C 180,E1 9123.131,E2 9123.131} C_VEL
LIN {X 0,Y 200.77,Z 1045.311,A -85,B 0,C 180,E1 9115.993,E2 9115.993} C_VEL
LIN {X 0,Y 196.396,Z 1050.161,A -85,B 0,C 180,E1 9109.944,E2 9109.944} C_VEL
LIN {X 0,Y 193.66,Z 1053.895,A -85,B 0,C 180,E1 9103.739,E2 9103.739} C_VEL
LIN {X 0,Y 192.277,Z 1056.659,A -85,B 0,C 180,E1 9097.169,E2 9097.169} C_VEL
LIN {X 0,Y 191.95,Z 1058.24,A -85,B 0,C 180,E1 9090.597,E2 9090.597} C_VEL
LIN {X 0,Y 191.922,Z 1058.592,A -85,B 0,C 180,E1 9084.619,E2 9084.619} C_VEL
LIN {X 0,Y 192.132,Z 1057.975,A -85,B 0,C 180,E1 9078.594,E2 9078.594} C_VEL
LIN {X 0,Y 193.149,Z 1056.264,A -85,B 0,C 180,E1 9072.216,E2 9072.216} C_VEL
LIN {X 0,Y 195.391,Z 1053.62,A -85,B 0,C 180,E1 9066.154,E2 9066.154} C_VEL
LIN {X 0,Y 199.374,Z 1049.743,A -85,B 0,C 180,E1 9059.9,E2 9059.9} C_VEL
LIN {X 0,Y 206.925,Z 1043.277,A -85,B 0,C 180,E1 9052.417,E2 9052.417} C_VEL
LIN {X 0,Y 215.884,Z 1035.895,A -85,B 0,C 180,E1 9046.264,E2 9046.264} C_VEL
LIN {X 0,Y 226.249,Z 1027.555,A -85,B 0,C 180,E1 9040.912,E2 9040.912} C_VEL
LIN {X 0,Y 240.198,Z 1016.053,A -85,B 0,C 180,E1 9035.324,E2 9035.324} C_VEL
LIN {X 0,Y 252.757,Z 1005.249,A -85,B 0,C 180,E1 9031.298,E2 9031.298} C_VEL
LIN {X 0,Y 266.407,Z 992.975,A -85,B 0,C 180,E1 9027.655,E2 9027.655} C_VEL
LIN {X 0,Y 282.813,Z 977.095,A -85,B 0,C 180,E1 9023.991,E2 9023.991} C_VEL
LIN {X 0,Y 295.61,Z 963.745,A -85,B 0,C 180,E1 9021.538,E2 9021.538} C_VEL
LIN {X 0,Y 309.234,Z 948.5,A -85,B 0,C 180,E1 9019.238,E2 9019.238} C_VEL
LIN {X 0,Y 325.841,Z 928.073,A -85,B 0,C 180,E1 9016.782,E2 9016.782} C_VEL
LIN {X 0,Y 338.215,Z 911.234,A -85,B 0,C 180,E1 9015.149,E2 9015.149} C_VEL
LIN {X 0,Y 351.076,Z 892.059,A -85,B 0,C 180,E1 9013.609,E2 9013.609} C_VEL
LIN {X 0,Y 364.621,Z 869.223,A -85,B 0,C 180,E1 9012.134,E2 9012.134} C_VEL
LIN {X 0,Y 374.517,Z 850.421,A -85,B 0,C 180,E1 9011.143,E2 9011.143} C_VEL
LIN {X 0,Y 384.07,Z 830.028,A -85,B 0,C 180,E1 9010.237,E2 9010.237} C_VEL
LIN {X 0,Y 394.174,Z 804.841,A -85,B 0,C 180,E1 9009.334,E2 9009.334} C_VEL
LIN {X 0,Y 401.328,Z 783.657,A -85,B 0,C 180,E1 9008.729,E2 9008.729} C_VEL
LIN {X 0,Y 407.29,Z 762.731,A -85,B 0,C 180,E1 9008.247,E2 9008.247} C_VEL
LIN {X 0,Y 413.503,Z 734.848,A -85,B 0,C 180,E1 9007.742,E2 9007.742} C_VEL
LIN {X 0,Y 417.115,Z 711.996,A -85,B 0,C 180,E1 9007.402,E2 9007.402} C_VEL
LIN {X 0,Y 433.619,Z 563.802,A -85,B 0,C 180,E1 9005.392,E2 9005.392} C_VEL
LIN {X 0,Y 432.514,Z 561.166,A -85,B 0,C 180,E1 9003.579,E2 9003.579} C_VEL
LIN {X 0,Y 431.384,Z 557.492,A -85,B 0,C 180,E1 8999.734,E2 8999.734} C_VEL
LIN {X 0,Y 431.366,Z 557.523,A -85,B 0,C 180,E1 8997.445,E2 8997.445} C_VEL
LIN {X 0,Y 431.419,Z 558.53,A -85,B 0,C 180,E1 8996.579,E2 8996.579} C_VEL
LIN {X 0,Y 431.383,Z 562.246,A -85,B 0,C 180,E1 8995.348,E2 8995.348} C_VEL
LIN {X 0,Y 431.566,Z 568.476,A -85,B 0,C 180,E1 8993.586,E2 8993.586} C_VEL
LIN {X 0,Y 431.806,Z 569.748,A -85,B 0,C 180,E1 8993.014,E2 8993.014} C_VEL
LIN {X 0,Y 432.007,Z 570.477,A -85,B 0,C 180,E1 8992.631,E2 8992.631} C_VEL
LIN {X 0,Y 415.389,Z 716.606,A -85,B 0,C 180,E1 8990.693,E2 8990.693} C_VEL
LIN {X 0,Y 410.593,Z 744.109,A -85,B 0,C 180,E1 8990.284,E2 8990.284} C_VEL
LIN {X 0,Y 405.101,Z 766.892,A -85,B 0,C 180,E1 8989.879,E2 8989.879} C_VEL
LIN {X 0,Y 398.743,Z 788.394,A -85,B 0,C 180,E1 8989.413,E2 8989.413} C_VEL
LIN {X 0,Y 389.258,Z 814.824,A -85,B 0,C 180,E1 8988.664,E2 8988.664} C_VEL
LIN {X 0,Y 380.382,Z 835.635,A -85,B 0,C 180,E1 8987.919,E2 8987.919} C_VEL
LIN {X 0,Y 371.306,Z 854.418,A -85,B 0,C 180,E1 8987.116,E2 8987.116} C_VEL
LIN {X 0,Y 358.744,Z 877.431,A -85,B 0,C 180,E1 8985.916,E2 8985.916} C_VEL
LIN {X 0,Y 345.9,Z 897.959,A -85,B 0,C 180,E1 8984.577,E2 8984.577} C_VEL
LIN {X 0,Y 333.863,Z 915.411,A -85,B 0,C 180,E1 8983.195,E2 8983.195} C_VEL
LIN {X 0,Y 318.393,Z 935.71,A -85,B 0,C 180,E1 8981.223,E2 8981.223} C_VEL
LIN {X 0,Y 303.893,Z 952.795,A -85,B 0,C 180,E1 8979.137,E2 8979.137} C_VEL
LIN {X 0,Y 289.851,Z 968.087,A -85,B 0,C 180,E1 8976.842,E2 8976.842} C_VEL
LIN {X 0,Y 272.515,Z 985.412,A -85,B 0,C 180,E1 8973.542,E2 8973.542} C_VEL
LIN {X 0,Y 258.665,Z 998.179,A -85,B 0,C 180,E1 8970.43,E2 8970.43} C_VEL
LIN {X 0,Y 244.988,Z 1010.108,A -85,B 0,C 180,E1 8966.791,E2 8966.791} C_VEL
LIN {X 0,Y 229.392,Z 1022.95,A -85,B 0,C 180,E1 8961.683,E2 8961.683} C_VEL
LIN {X 0,Y 217.573,Z 1032.293,A -85,B 0,C 180,E1 8956.783,E2 8956.783} C_VEL
LIN {X 0,Y 206.721,Z 1040.816,A -85,B 0,C 180,E1 8951.013,E2 8951.013} C_VEL
LIN {X 0,Y 197.031,Z 1048.501,A -85,B 0,C 180,E1 8943.933,E2 8943.933} C_VEL
LIN {X 0,Y 190.923,Z 1053.681,A -85,B 0,C 180,E1 8937.443,E2 8937.443} C_VEL
LIN {X 0,Y 186.866,Z 1057.643,A -85,B 0,C 180,E1 8930.68,E2 8930.68} C_VEL
LIN {X 0,Y 184.483,Z 1060.722,A -85,B 0,C 180,E1 8922.684,E2 8922.684} C_VEL
LIN {X 0,Y 183.939,Z 1061.958,A -85,B 0,C 180,E1 8916.242,E2 8916.242} C_VEL
LIN {X 0,Y 183.92,Z 1062.212,A -85,B 0,C 180,E1 8910.623,E2 8910.623} C_VEL
LIN {X 0,Y 183.913,Z 1061.648,A -85,B 0,C 180,E1 8905.01,E2 8905.01} C_VEL
LIN {X 0,Y 184.263,Z 1060.031,A -85,B 0,C 180,E1 8898.735,E2 8898.735} C_VEL
LIN {X 0,Y 185.605,Z 1057.397,A -85,B 0,C 180,E1 8892.442,E2 8892.442} C_VEL
LIN {X 0,Y 188.34,Z 1053.729,A -85,B 0,C 180,E1 8886.204,E2 8886.204} C_VEL
LIN {X 0,Y 192.959,Z 1048.741,A -85,B 0,C 180,E1 8879.825,E2 8879.825} C_VEL
LIN {X 0,Y 201.265,Z 1040.882,A -85,B 0,C 180,E1 8872.334,E2 8872.334} C_VEL
LIN {X 0,Y 210.448,Z 1032.598,A -85,B 0,C 180,E1 8866.455,E2 8866.455} C_VEL
LIN {X 0,Y 220.937,Z 1023.337,A -85,B 0,C 180,E1 8861.301,E2 8861.301} C_VEL
LIN {X 0,Y 235.353,Z 1010.339,A -85,B 0,C 180,E1 8855.762,E2 8855.762} C_VEL
LIN {X 0,Y 247.798,Z 998.616,A -85,B 0,C 180,E1 8851.911,E2 8851.911} C_VEL
LIN {X 0,Y 261.399,Z 985.213,A -85,B 0,C 180,E1 8848.385,E2 8848.385} C_VEL
LIN {X 0,Y 277.666,Z 967.953,A -85,B 0,C 180,E1 8844.843,E2 8844.843} C_VEL
LIN {X 0,Y 290.867,Z 952.805,A -85,B 0,C 180,E1 8842.375,E2 8842.375} C_VEL
LIN {X 0,Y 305.798,Z 934.36,A -85,B 0,C 180,E1 8839.94,E2 8839.94} C_VEL
LIN {X 0,Y 319.946,Z 914.808,A -85,B 0,C 180,E1 8837.897,E2 8837.897} C_VEL
LIN {X 0,Y 331.685,Z 897.051,A -85,B 0,C 180,E1 8836.373,E2 8836.373} C_VEL
LIN {X 0,Y 344.496,Z 875.693,A -85,B 0,C 180,E1 8834.869,E2 8834.869} C_VEL
LIN {X 0,Y 355.982,Z 853.708,A -85,B 0,C 180,E1 8833.628,E2 8833.628} C_VEL
LIN {X 0,Y 364.924,Z 834.484,A -85,B 0,C 180,E1 8832.727,E2 8832.727} C_VEL
LIN {X 0,Y 374.868,Z 810.055,A -85,B 0,C 180,E1 8831.792,E2 8831.792} C_VEL
LIN {X 0,Y 382.823,Z 786.417,A -85,B 0,C 180,E1 8831.083,E2 8831.083} C_VEL
LIN {X 0,Y 388.793,Z 765.397,A -85,B 0,C 180,E1 8830.588,E2 8830.588} C_VEL
LIN {X 0,Y 394.691,Z 739.444,A -85,B 0,C 180,E1 8830.096,E2 8830.096} C_VEL
LIN {X 0,Y 398.63,Z 714.588,A -85,B 0,C 180,E1 8829.707,E2 8829.707} C_VEL
LIN {X 0,Y 415.743,Z 556.814,A -85,B 0,C 180,E1 8827.507,E2 8827.507} C_VEL
LIN {X 0,Y 413.878,Z 552.658,A -85,B 0,C 180,E1 8825.128,E2 8825.128} C_VEL
LIN {X 0,Y 412.613,Z 549.619,A -85,B 0,C 180,E1 8822.778,E2 8822.778} C_VEL
LIN {X 0,Y 411.711,Z 547.281,A -85,B 0,C 180,E1 8818.191,E2 8818.191} C_VEL
LIN {X 0,Y 412.88,Z 550.19,A -85,B 0,C 180,E1 8813.464,E2 8813.464} C_VEL
LIN {X 0,Y 414.584,Z 554.246,A -85,B 0,C 180,E1 8810.701,E2 8810.701} C_VEL
LIN {X 0,Y 415.736,Z 556.863,A -85,B 0,C 180,E1 8809.314,E2 8809.314} C_VEL
LIN {X 0,Y 398.483,Z 715.194,A -85,B 0,C 180,E1 8807.129,E2 8807.129} C_VEL
LIN {X 0,Y 393.875,Z 742.516,A -85,B 0,C 180,E1 8806.692,E2 8806.692} C_VEL
LIN {X 0,Y 388.412,Z 765.836,A -85,B 0,C 180,E1 8806.223,E2 8806.223} C_VEL
LIN {X 0,Y 382.56,Z 786.315,A -85,B 0,C 180,E1 8805.7,E2 8805.7} C_VEL
LIN {X 0,Y 373.867,Z 811.618,A -85,B 0,C 180,E1 8804.9,E2 8804.9} C_VEL
LIN {X 0,Y 365.019,Z 833.143,A -85,B 0,C 180,E1 8804.046,E2 8804.046} C_VEL
LIN {X 0,Y 355.837,Z 852.844,A -85,B 0,C 180,E1 8803.095,E2 8803.095} C_VEL
LIN {X 0,Y 344.177,Z 875.022,A -85,B 0,C 180,E1 8801.802,E2 8801.802} C_VEL
LIN {X 0,Y 331.838,Z 895.501,A -85,B 0,C 180,E1 8800.324,E2 8800.324} C_VEL
LIN {X 0,Y 320.154,Z 913.121,A -85,B 0,C 180,E1 8798.789,E2 8798.789} C_VEL
LIN {X 0,Y 305.806,Z 932.825,A -85,B 0,C 180,E1 8796.694,E2 8796.694} C_VEL
LIN {X 0,Y 291.668,Z 950.248,A -85,B 0,C 180,E1 8794.37,E2 8794.37} C_VEL
LIN {X 0,Y 278.715,Z 965.07,A -85,B 0,C 180,E1 8791.948,E2 8791.948} C_VEL
LIN {X 0,Y 262.742,Z 982.021,A -85,B 0,C 180,E1 8788.479,E2 8788.479} C_VEL
LIN {X 0,Y 249.086,Z 995.404,A -85,B 0,C 180,E1 8784.968,E2 8784.968} C_VEL
LIN {X 0,Y 236.433,Z 1007.229,A -85,B 0,C 180,E1 8781.091,E2 8781.091} C_VEL
LIN {X 0,Y 221.637,Z 1020.419,A -85,B 0,C 180,E1 8775.462,E2 8775.462} C_VEL
LIN {X 0,Y 211.277,Z 1029.431,A -85,B 0,C 180,E1 8770.418,E2 8770.418} C_VEL
LIN {X 0,Y 201.75,Z 1037.845,A -85,B 0,C 180,E1 8764.401,E2 8764.401} C_VEL
LIN {X 0,Y 193.47,Z 1045.449,A -85,B 0,C 180,E1 8757.052,E2 8757.052} C_VEL
LIN {X 0,Y 188.78,Z 1050.287,A -85,B 0,C 180,E1 8750.785,E2 8750.785} C_VEL
LIN {X 0,Y 185.82,Z 1054.011,A -85,B 0,C 180,E1 8744.331,E2 8744.331} C_VEL
LIN {X 0,Y 184.275,Z 1056.875,A -85,B 0,C 180,E1 8737.169,E2 8737.169} C_VEL
LIN {X 0,Y 183.948,Z 1058.345,A -85,B 0,C 180,E1 8730.311,E2 8730.311} C_VEL
LIN {X 0,Y 183.933,Z 1058.643,A -85,B 0,C 180,E1 8724.071,E2 8724.071} C_VEL
LIN {X 0,Y 184.202,Z 1057.957,A -85,B 0,C 180,E1 8717.71,E2 8717.71} C_VEL
LIN {X 0,Y 185.333,Z 1056.318,A -85,B 0,C 180,E1 8711.439,E2 8711.439} C_VEL
LIN {X 0,Y 187.822,Z 1053.663,A -85,B 0,C 180,E1 8705.13,E2 8705.13} C_VEL
LIN {X 0,Y 192.303,Z 1049.681,A -85,B 0,C 180,E1 8698.51,E2 8698.51} C_VEL
LIN {X 0,Y 200.613,Z 1043.051,A -85,B 0,C 180,E1 8690.729,E2 8690.729} C_VEL
LIN {X 0,Y 209.75,Z 1035.987,A -85,B 0,C 180,E1 8684.742,E2 8684.742} C_VEL
LIN {X 0,Y 220.416,Z 1027.836,A -85,B 0,C 180,E1 8679.427,E2 8679.427} C_VEL
LIN {X 0,Y 235.419,Z 1016.014,A -85,B 0,C 180,E1 8673.647,E2 8673.647} C_VEL
LIN {X 0,Y 248.484,Z 1005.196,A -85,B 0,C 180,E1 8669.637,E2 8669.637} C_VEL
LIN {X 0,Y 262.61,Z 992.909,A -85,B 0,C 180,E1 8666.029,E2 8666.029} C_VEL
LIN {X 0,Y 279.186,Z 977.316,A -85,B 0,C 180,E1 8662.481,E2 8662.481} C_VEL
LIN {X 0,Y 293.005,Z 963.25,A -85,B 0,C 180,E1 8659.953,E2 8659.953} C_VEL
LIN {X 0,Y 307.008,Z 947.902,A -85,B 0,C 180,E1 8657.705,E2 8657.705} C_VEL
LIN {X 0,Y 323.542,Z 927.903,A -85,B 0,C 180,E1 8655.374,E2 8655.374} C_VEL
LIN {X 0,Y 335.709,Z 911.653,A -85,B 0,C 180,E1 8653.84,E2 8653.84} C_VEL
LIN {X 0,Y 348.101,Z 893.533,A -85,B 0,C 180,E1 8652.415,E2 8652.415} C_VEL
LIN {X 0,Y 362.515,Z 869.782,A -85,B 0,C 180,E1 8650.913,E2 8650.913} C_VEL
LIN {X 0,Y 372.562,Z 851.006,A -85,B 0,C 180,E1 8649.95,E2 8649.95} C_VEL
LIN {X 0,Y 381.776,Z 831.686,A -85,B 0,C 180,E1 8649.113,E2 8649.113} C_VEL
LIN {X 0,Y 392.002,Z 806.941,A -85,B 0,C 180,E1 8648.24,E2 8648.24} C_VEL
LIN {X 0,Y 399.655,Z 784.733,A -85,B 0,C 180,E1 8647.62,E2 8647.62} C_VEL
LIN {X 0,Y 405.556,Z 764.448,A -85,B 0,C 180,E1 8647.163,E2 8647.163} C_VEL
LIN {X 0,Y 411.598,Z 738.748,A -85,B 0,C 180,E1 8646.7,E2 8646.7} C_VEL
LIN {X 0,Y 415.767,Z 713.375,A -85,B 0,C 180,E1 8646.328,E2 8646.328} C_VEL
LIN {X 0,Y 431.984,Z 570.364,A -85,B 0,C 180,E1 8644.417,E2 8644.417} C_VEL
LIN {X 0,Y 431.322,Z 568.815,A -85,B 0,C 180,E1 8643.189,E2 8643.189} C_VEL
LIN {X 0,Y 430.409,Z 565.433,A -85,B 0,C 180,E1 8639.734,E2 8639.734} C_VEL
LIN {X 0,Y 430.456,Z 565.68,A -85,B 0,C 180,E1 8636.937,E2 8636.937} C_VEL
LIN {X 0,Y 431.806,Z 569.748,A -85,B 0,C 180,E1 8633.014,E2 8633.014} C_VEL
LIN {X 0,Y 431.781,Z 571.262,A -85,B 0,C 180,E1 8632.798,E2 8632.798} C_VEL
LIN {X 0,Y 431.456,Z 574.36,A -85,B 0,C 180,E1 8632.723,E2 8632.723} C_VEL
LIN {X 0,Y 430.753,Z 579.241,A -85,B 0,C 180,E1 8632.855,E2 8632.855} C_VEL
LIN {X 0,Y 429.22,Z 588.816,A -85,B 0,C 180,E1 8633.345,E2 8633.345} C_VEL
LIN {X 0,Y 428.623,Z 593.36,A -85,B 0,C 180,E1 8633.398,E2 8633.398} C_VEL
LIN {X 0,Y 414.346,Z 716.726,A -85,B 0,C 180,E1 8631.791,E2 8631.791} C_VEL
LIN {X 0,Y 409.412,Z 744.5,A -85,B 0,C 180,E1 8631.389,E2 8631.389} C_VEL
LIN {X 0,Y 403.923,Z 766.988,A -85,B 0,C 180,E1 8631.004,E2 8631.004} C_VEL
LIN {X 0,Y 397.353,Z 788.925,A -85,B 0,C 180,E1 8630.545,E2 8630.545} C_VEL
LIN {X 0,Y 387.477,Z 815.9,A -85,B 0,C 180,E1 8629.804,E2 8629.804} C_VEL
LIN {X 0,Y 378.782,Z 835.972,A -85,B 0,C 180,E1 8629.107,E2 8629.107} C_VEL
LIN {X 0,Y 368.873,Z 856.124,A -85,B 0,C 180,E1 8628.27,E2 8628.27} C_VEL
LIN {X 0,Y 355.505,Z 879.849,A -85,B 0,C 180,E1 8627.047,E2 8627.047} C_VEL
LIN {X 0,Y 343.401,Z 898.799,A -85,B 0,C 180,E1 8625.836,E2 8625.836} C_VEL
LIN {X 0,Y 330.6,Z 916.968,A -85,B 0,C 180,E1 8624.427,E2 8624.427} C_VEL
LIN {X 0,Y 314.035,Z 937.984,A -85,B 0,C 180,E1 8622.393,E2 8622.393} C_VEL
LIN {X 0,Y 301.066,Z 952.91,A -85,B 0,C 180,E1 8620.597,E2 8620.597} C_VEL
LIN {X 0,Y 287.091,Z 967.786,A -85,B 0,C 180,E1 8618.421,E2 8618.421} C_VEL
LIN {X 0,Y 268.932,Z 985.477,A -85,B 0,C 180,E1 8615.12,E2 8615.12} C_VEL
LIN {X 0,Y 254.676,Z 998.231,A -85,B 0,C 180,E1 8612.052,E2 8612.052} C_VEL
LIN {X 0,Y 240.298,Z 1010.349,A -85,B 0,C 180,E1 8608.379,E2 8608.379} C_VEL
LIN {X 0,Y 224.161,Z 1023.088,A -85,B 0,C 180,E1 8603.293,E2 8603.293} C_VEL
LIN {X 0,Y 212.179,Z 1032.125,A -85,B 0,C 180,E1 8598.528,E2 8598.528} C_VEL
LIN {X 0,Y 200.67,Z 1040.692,A -85,B 0,C 180,E1 8592.66,E2 8592.66} C_VEL
LIN {X 0,Y 190.207,Z 1048.473,A -85,B 0,C 180,E1 8585.328,E2 8585.328} C_VEL
LIN {X 0,Y 183.635,Z 1053.643,A -85,B 0,C 180,E1 8578.631,E2 8578.631} C_VEL
LIN {X 0,Y 179.21,Z 1057.595,A -85,B 0,C 180,E1 8571.607,E2 8571.607} C_VEL
LIN {X 0,Y 176.599,Z 1060.623,A -85,B 0,C 180,E1 8563.423,E2 8563.423} C_VEL
LIN {X 0,Y 175.95,Z 1061.885,A -85,B 0,C 180,E1 8556.526,E2 8556.526} C_VEL
LIN {X 0,Y 175.92,Z 1062.129,A -85,B 0,C 180,E1 8550.651,E2 8550.651} C_VEL
LIN {X 0,Y 175.916,Z 1061.556,A -85,B 0,C 180,E1 8544.782,E2 8544.782} C_VEL
LIN {X 0,Y 176.321,Z 1059.929,A -85,B 0,C 180,E1 8538.22,E2 8538.22} C_VEL
LIN {X 0,Y 177.824,Z 1057.285,A -85,B 0,C 180,E1 8531.647,E2 8531.647} C_VEL
LIN {X 0,Y 180.91,Z 1053.519,A -85,B 0,C 180,E1 8525.017,E2 8525.017} C_VEL
LIN {X 0,Y 186.43,Z 1048.092,A -85,B 0,C 180,E1 8517.929,E2 8517.929} C_VEL
LIN {X 0,Y 195.545,Z 1040.011,A -85,B 0,C 180,E1 8510.271,E2 8510.271} C_VEL
LIN {X 0,Y 204.964,Z 1032.022,A -85,B 0,C 180,E1 8504.583,E2 8504.583} C_VEL
LIN {X 0,Y 216.651,Z 1022.23,A -85,B 0,C 180,E1 8499.163,E2 8499.163} C_VEL
LIN {X 0,Y 231.206,Z 1009.556,A -85,B 0,C 180,E1 8493.868,E2 8493.868} C_VEL
LIN {X 0,Y 243.92,Z 997.998,A -85,B 0,C 180,E1 8490.125,E2 8490.125} C_VEL
LIN {X 0,Y 258.283,Z 984.275,A -85,B 0,C 180,E1 8486.586,E2 8486.586} C_VEL
LIN {X 0,Y 274.277,Z 967.694,A -85,B 0,C 180,E1 8483.267,E2 8483.267} C_VEL
LIN {X 0,Y 287.813,Z 952.53,A -85,B 0,C 180,E1 8480.849,E2 8480.849} C_VEL
LIN {X 0,Y 303.154,Z 933.966,A -85,B 0,C 180,E1 8478.46,E2 8478.46} C_VEL
LIN {X 0,Y 317.079,Z 915.086,A -85,B 0,C 180,E1 8476.537,E2 8476.537} C_VEL
LIN {X 0,Y 328.894,Z 897.562,A -85,B 0,C 180,E1 8475.067,E2 8475.067} C_VEL
LIN {X 0,Y 342.038,Z 876.08,A -85,B 0,C 180,E1 8473.591,E2 8473.591} C_VEL
LIN {X 0,Y 353.692,Z 854.16,A -85,B 0,C 180,E1 8472.387,E2 8472.387} C_VEL
LIN {X 0,Y 362.759,Z 834.998,A -85,B 0,C 180,E1 8471.514,E2 8471.514} C_VEL
LIN {X 0,Y 372.696,Z 811.095,A -85,B 0,C 180,E1 8470.622,E2 8470.622} C_VEL
LIN {X 0,Y 381.04,Z 786.707,A -85,B 0,C 180,E1 8469.911,E2 8469.911} C_VEL
LIN {X 0,Y 387.149,Z 765.487,A -85,B 0,C 180,E1 8469.428,E2 8469.428} C_VEL
LIN {X 0,Y 393.091,Z 739.757,A -85,B 0,C 180,E1 8468.956,E2 8468.956} C_VEL
LIN {X 0,Y 397.14,Z 714.592,A -85,B 0,C 180,E1 8468.572,E2 8468.572} C_VEL
LIN {X 0,Y 413.867,Z 563.117,A -85,B 0,C 180,E1 8466.503,E2 8466.503} C_VEL
LIN {X 0,Y 412.617,Z 560.185,A -85,B 0,C 180,E1 8464.726,E2 8464.726} C_VEL
LIN {X 0,Y 411.57,Z 557.502,A -85,B 0,C 180,E1 8462.646,E2 8462.646} C_VEL
LIN {X 0,Y 410.735,Z 555.232,A -85,B 0,C 180,E1 8458.186,E2 8458.186} C_VEL
LIN {X 0,Y 411.8,Z 557.997,A -85,B 0,C 180,E1 8453.657,E2 8453.657} C_VEL
LIN {X 0,Y 413.388,Z 561.941,A -85,B 0,C 180,E1 8450.954,E2 8450.954} C_VEL
LIN {X 0,Y 413.839,Z 563.292,A -85,B 0,C 180,E1 8450.324,E2 8450.324} C_VEL
LIN {X 0,Y 396.989,Z 715.273,A -85,B 0,C 180,E1 8448.263,E2 8448.263} C_VEL
LIN {X 0,Y 392.343,Z 742.501,A -85,B 0,C 180,E1 8447.84,E2 8447.84} C_VEL
LIN {X 0,Y 386.794,Z 765.915,A -85,B 0,C 180,E1 8447.384,E2 8447.384} C_VEL
LIN {X 0,Y 380.896,Z 786.303,A -85,B 0,C 180,E1 8446.882,E2 8446.882} C_VEL
LIN {X 0,Y 372.315,Z 811.069,A -85,B 0,C 180,E1 8446.129,E2 8446.129} C_VEL
LIN {X 0,Y 362.9,Z 833.66,A -85,B 0,C 180,E1 8445.261,E2 8445.261} C_VEL
LIN {X 0,Y 353.588,Z 853.316,A -85,B 0,C 180,E1 8444.338,E2 8444.338} C_VEL
LIN {X 0,Y 341.416,Z 875.977,A -85,B 0,C 180,E1 8443.047,E2 8443.047} C_VEL
LIN {X 0,Y 329.208,Z 895.873,A -85,B 0,C 180,E1 8441.647,E2 8441.647} C_VEL
LIN {X 0,Y 317.316,Z 913.47,A -85,B 0,C 180,E1 8440.151,E2 8440.151} C_VEL
LIN {X 0,Y 301.959,Z 934.021,A -85,B 0,C 180,E1 8437.998,E2 8437.998} C_VEL
LIN {X 0,Y 288.242,Z 950.535,A -85,B 0,C 180,E1 8435.828,E2 8435.828} C_VEL
LIN {X 0,Y 274.798,Z 965.533,A -85,B 0,C 180,E1 8433.413,E2 8433.413} C_VEL
LIN {X 0,Y 258.56,Z 982.259,A -85,B 0,C 180,E1 8430.024,E2 8430.024} C_VEL
LIN {X 0,Y 244.487,Z 995.618,A -85,B 0,C 180,E1 8426.543,E2 8426.543} C_VEL
LIN {X 0,Y 231.371,Z 1007.44,A -85,B 0,C 180,E1 8422.671,E2 8422.671} C_VEL
LIN {X 0,Y 216.521,Z 1020.151,A -85,B 0,C 180,E1 8417.244,E2 8417.244} C_VEL
LIN {X 0,Y 205.581,Z 1029.204,A -85,B 0,C 180,E1 8412.159,E2 8412.159} C_VEL
LIN {X 0,Y 195.843,Z 1037.31,A -85,B 0,C 180,E1 8406.316,E2 8406.316} C_VEL
LIN {X 0,Y 186.457,Z 1045.397,A -85,B 0,C 180,E1 8398.422,E2 8398.422} C_VEL
LIN {X 0,Y 181.205,Z 1050.413,A -85,B 0,C 180,E1 8391.697,E2 8391.697} C_VEL
LIN {X 0,Y 177.981,Z 1054.153,A -85,B 0,C 180,E1 8384.918,E2 8384.918} C_VEL
LIN {X 0,Y 176.272,Z 1057.091,A -85,B 0,C 180,E1 8377.169,E2 8377.169} C_VEL
LIN {X 0,Y 175.946,Z 1058.451,A -85,B 0,C 180,E1 8370,E2 8370} C_VEL
LIN {X 0,Y 175.937,Z 1058.716,A -85,B 0,C 180,E1 8363.801,E2 8363.801} C_VEL
LIN {X 0,Y 176.23,Z 1058.071,A -85,B 0,C 180,E1 8357.395,E2 8357.395} C_VEL
LIN {X 0,Y 177.547,Z 1056.371,A -85,B 0,C 180,E1 8350.593,E2 8350.593} C_VEL
LIN {X 0,Y 180.373,Z 1053.65,A -85,B 0,C 180,E1 8343.902,E2 8343.902} C_VEL
LIN {X 0,Y 185.37,Z 1049.603,A -85,B 0,C 180,E1 8336.989,E2 8336.989} C_VEL
LIN {X 0,Y 194.564,Z 1042.758,A -85,B 0,C 180,E1 8328.867,E2 8328.867} C_VEL
LIN {X 0,Y 204.224,Z 1035.756,A -85,B 0,C 180,E1 8322.887,E2 8322.887} C_VEL
LIN {X 0,Y 216.128,Z 1027.122,A -85,B 0,C 180,E1 8317.275,E2 8317.275} C_VEL
LIN {X 0,Y 230.878,Z 1015.953,A -85,B 0,C 180,E1 8311.895,E2 8311.895} C_VEL
LIN {X 0,Y 244.427,Z 1005.145,A -85,B 0,C 180,E1 8307.92,E2 8307.92} C_VEL
LIN {X 0,Y 259.785,Z 992.205,A -85,B 0,C 180,E1 8304.191,E2 8304.191} C_VEL
LIN {X 0,Y 276.836,Z 976.488,A -85,B 0,C 180,E1 8300.73,E2 8300.73} C_VEL
LIN {X 0,Y 290.713,Z 962.667,A -85,B 0,C 180,E1 8298.326,E2 8298.326} C_VEL
LIN {X 0,Y 306.716,Z 945.442,A -85,B 0,C 180,E1 8295.91,E2 8295.91} C_VEL
LIN {X 0,Y 322.319,Z 926.614,A -85,B 0,C 180,E1 8293.838,E2 8293.838} C_VEL
LIN {X 0,Y 334.961,Z 909.907,A -85,B 0,C 180,E1 8292.335,E2 8292.335} C_VEL
LIN {X 0,Y 349.152,Z 889.233,A -85,B 0,C 180,E1 8290.806,E2 8290.806} C_VEL
LIN {X 0,Y 362.045,Z 867.729,A -85,B 0,C 180,E1 8289.538,E2 8289.538} C_VEL
LIN {X 0,Y 372.492,Z 848.225,A -85,B 0,C 180,E1 8288.592,E2 8288.592} C_VEL
LIN {X 0,Y 383.388,Z 825.084,A -85,B 0,C 180,E1 8287.672,E2 8287.672} C_VEL
LIN {X 0,Y 392.336,Z 802.562,A -85,B 0,C 180,E1 8286.948,E2 8286.948} C_VEL
LIN {X 0,Y 399.444,Z 781.68,A -85,B 0,C 180,E1 8286.4,E2 8286.4} C_VEL
LIN {X 0,Y 406.624,Z 756.198,A -85,B 0,C 180,E1 8285.881,E2 8285.881} C_VEL
LIN {X 0,Y 411.839,Z 731.554,A -85,B 0,C 180,E1 8285.486,E2 8285.486} C_VEL
LIN {X 0,Y 415.36,Z 708.896,A -85,B 0,C 180,E1 8285.169,E2 8285.169} C_VEL
LIN {X 0,Y 430.464,Z 577,A -85,B 0,C 180,E1 8283.429,E2 8283.429} C_VEL
LIN {X 0,Y 429.415,Z 573.358,A -85,B 0,C 180,E1 8279.6,E2 8279.6} C_VEL
